(* Logix 5000 project; controller QW361 vendor 1 type 14 code 107 rev 32.11; software revision 32.00; part 13 of 20 *)

        [1807].time.Minute := 9, [1807].time.Second := 59, [1807].time.DST_ON := 1, [1808].log_data[0].min := 1.0, [1808].log_data[0].max := 1.0, [1808].log_data[0].total := 300.0, [1808].log_data[0].time := 300.0, [1808].log_data[0].minminute := 10, [1808].log_data[0].maxminute := 10, [1808].log_data[0].valid := 1, [1808].log_data[1].valid := 1, [1808].log_data[2].valid := 1, [1808].log_data[3].valid := 1, [1808].log_data[4].valid := 1, [1808].time.Year := 2022, [1808].time.Month := 4, [1808].time.Day := 30, [1808].time.Hour := 4, [1808].time.Minute := 14, [1808].time.Second := 59, [1808].time.DST_ON := 1, [1809].log_data[0].min := 1.0, [1809].log_data[0].max := 1.0, [1809].log_data[0].total := 300.0, [1809].log_data[0].time := 300.0, [1809].log_data[0].minminute := 15, [1809].log_data[0].maxminute := 15, [1809].log_data[0].valid := 1, [1809].log_data[1].valid := 1, [1809].log_data[2].valid := 1, [1809].log_data[3].valid := 1, [1809].log_data[4].valid := 1, [1809].time.Year := 2022, [1809].time.Month := 4, [1809].time.Day := 30, [1809].time.Hour := 4, [1809].time.Minute := 19, [1809].time.Second := 59, [1809].time.DST_ON := 1, [1810].log_data[0].min := 1.0, [1810].log_data[0].max := 1.0, [1810].log_data[0].total := 300.0, [1810].log_data[0].time := 300.0, [1810].log_data[0].minminute := 20, [1810].log_data[0].maxminute := 20, [1810].log_data[0].valid := 1, [1810].log_data[1].valid := 1, [1810].log_data[2].valid := 1, [1810].log_data[3].valid := 1, [1810].log_data[4].valid := 1, [1810].time.Year := 2022, [1810].time.Month := 4, [1810].time.Day := 30, [1810].time.Hour := 4, [1810].time.Minute := 24, [1810].time.Second := 59, [1810].time.DST_ON := 1, [1811].log_data[0].min := 1.0, [1811].log_data[0].max := 1.0, [1811].log_data[0].total := 300.0,
        [1811].log_data[0].time := 300.0, [1811].log_data[0].minminute := 25, [1811].log_data[0].maxminute := 25, [1811].log_data[0].valid := 1, [1811].log_data[1].valid := 1, [1811].log_data[2].valid := 1, [1811].log_data[3].valid := 1, [1811].log_data[4].valid := 1, [1811].time.Year := 2022, [1811].time.Month := 4, [1811].time.Day := 30, [1811].time.Hour := 4, [1811].time.Minute := 29, [1811].time.Second := 59, [1811].time.DST_ON := 1, [1812].log_data[0].min := 1.0, [1812].log_data[0].max := 1.0, [1812].log_data[0].total := 300.0, [1812].log_data[0].time := 300.0, [1812].log_data[0].minminute := 30, [1812].log_data[0].maxminute := 30, [1812].log_data[0].valid := 1, [1812].log_data[1].valid := 1, [1812].log_data[2].valid := 1, [1812].log_data[3].valid := 1, [1812].log_data[4].valid := 1, [1812].time.Year := 2022, [1812].time.Month := 4, [1812].time.Day := 30, [1812].time.Hour := 4, [1812].time.Minute := 34, [1812].time.Second := 59, [1812].time.DST_ON := 1, [1813].log_data[0].min := 1.0, [1813].log_data[0].max := 1.0, [1813].log_data[0].total := 300.0, [1813].log_data[0].time := 300.0, [1813].log_data[0].minminute := 35, [1813].log_data[0].maxminute := 35, [1813].log_data[0].valid := 1, [1813].log_data[1].valid := 1, [1813].log_data[2].valid := 1, [1813].log_data[3].valid := 1, [1813].log_data[4].valid := 1, [1813].time.Year := 2022, [1813].time.Month := 4, [1813].time.Day := 30, [1813].time.Hour := 4, [1813].time.Minute := 39, [1813].time.Second := 59, [1813].time.DST_ON := 1, [1814].log_data[0].min := 1.0, [1814].log_data[0].max := 1.0, [1814].log_data[0].total := 300.0, [1814].log_data[0].time := 300.0, [1814].log_data[0].minminute := 40, [1814].log_data[0].maxminute := 40, [1814].log_data[0].valid := 1, [1814].log_data[1].valid := 1, [1814].log_data[2].valid := 1,
        [1814].log_data[3].valid := 1, [1814].log_data[4].valid := 1, [1814].time.Year := 2022, [1814].time.Month := 4, [1814].time.Day := 30, [1814].time.Hour := 4, [1814].time.Minute := 44, [1814].time.Second := 59, [1814].time.DST_ON := 1, [1815].log_data[0].min := 1.0, [1815].log_data[0].max := 1.0, [1815].log_data[0].total := 300.0, [1815].log_data[0].time := 300.0, [1815].log_data[0].minminute := 45, [1815].log_data[0].maxminute := 45, [1815].log_data[0].valid := 1, [1815].log_data[1].valid := 1, [1815].log_data[2].valid := 1, [1815].log_data[3].valid := 1, [1815].log_data[4].valid := 1, [1815].time.Year := 2022, [1815].time.Month := 4, [1815].time.Day := 30, [1815].time.Hour := 4, [1815].time.Minute := 49, [1815].time.Second := 59, [1815].time.DST_ON := 1, [1816].log_data[0].min := 1.0, [1816].log_data[0].max := 1.0, [1816].log_data[0].total := 300.0, [1816].log_data[0].time := 300.0, [1816].log_data[0].minminute := 50, [1816].log_data[0].maxminute := 50, [1816].log_data[0].valid := 1, [1816].log_data[1].valid := 1, [1816].log_data[2].valid := 1, [1816].log_data[3].valid := 1, [1816].log_data[4].valid := 1, [1816].time.Year := 2022, [1816].time.Month := 4, [1816].time.Day := 30, [1816].time.Hour := 4, [1816].time.Minute := 54, [1816].time.Second := 59, [1816].time.DST_ON := 1, [1817].log_data[0].min := 1.0, [1817].log_data[0].max := 1.0, [1817].log_data[0].total := 300.0, [1817].log_data[0].time := 300.0, [1817].log_data[0].minminute := 55, [1817].log_data[0].maxminute := 55, [1817].log_data[0].valid := 1, [1817].log_data[1].valid := 1, [1817].log_data[2].valid := 1, [1817].log_data[3].valid := 1, [1817].log_data[4].valid := 1, [1817].time.Year := 2022, [1817].time.Month := 4, [1817].time.Day := 30, [1817].time.Hour := 4,
        [1817].time.Minute := 59, [1817].time.Second := 59, [1817].time.DST_ON := 1, [1818].log_data[0].min := 1.0, [1818].log_data[0].max := 1.0, [1818].log_data[0].total := 300.0, [1818].log_data[0].time := 300.0, [1818].log_data[0].valid := 1, [1818].log_data[1].valid := 1, [1818].log_data[2].valid := 1, [1818].log_data[3].valid := 1, [1818].log_data[4].valid := 1, [1818].time.Year := 2022, [1818].time.Month := 4, [1818].time.Day := 30, [1818].time.Hour := 5, [1818].time.Minute := 4, [1818].time.Second := 59, [1818].time.DST_ON := 1, [1819].log_data[0].min := 1.0, [1819].log_data[0].max := 1.0, [1819].log_data[0].total := 300.0, [1819].log_data[0].time := 300.0, [1819].log_data[0].minminute := 5, [1819].log_data[0].maxminute := 5, [1819].log_data[0].valid := 1, [1819].log_data[1].valid := 1, [1819].log_data[2].valid := 1, [1819].log_data[3].valid := 1, [1819].log_data[4].valid := 1, [1819].time.Year := 2022, [1819].time.Month := 4, [1819].time.Day := 30, [1819].time.Hour := 5, [1819].time.Minute := 9, [1819].time.Second := 59, [1819].time.DST_ON := 1, [1820].log_data[0].min := 1.0, [1820].log_data[0].max := 1.0, [1820].log_data[0].total := 300.0, [1820].log_data[0].time := 300.0, [1820].log_data[0].minminute := 10, [1820].log_data[0].maxminute := 10, [1820].log_data[0].valid := 1, [1820].log_data[1].valid := 1, [1820].log_data[2].valid := 1, [1820].log_data[3].valid := 1, [1820].log_data[4].valid := 1, [1820].time.Year := 2022, [1820].time.Month := 4, [1820].time.Day := 30, [1820].time.Hour := 5, [1820].time.Minute := 14, [1820].time.Second := 59, [1820].time.DST_ON := 1, [1821].log_data[0].min := 1.0, [1821].log_data[0].max := 1.0, [1821].log_data[0].total := 300.0, [1821].log_data[0].time := 300.0, [1821].log_data[0].minminute := 15,
        [1821].log_data[0].maxminute := 15, [1821].log_data[0].valid := 1, [1821].log_data[1].valid := 1, [1821].log_data[2].valid := 1, [1821].log_data[3].valid := 1, [1821].log_data[4].valid := 1, [1821].time.Year := 2022, [1821].time.Month := 4, [1821].time.Day := 30, [1821].time.Hour := 5, [1821].time.Minute := 19, [1821].time.Second := 59, [1821].time.DST_ON := 1, [1822].log_data[0].min := 1.0, [1822].log_data[0].max := 1.0, [1822].log_data[0].total := 300.0, [1822].log_data[0].time := 300.0, [1822].log_data[0].minminute := 20, [1822].log_data[0].maxminute := 20, [1822].log_data[0].valid := 1, [1822].log_data[1].valid := 1, [1822].log_data[2].valid := 1, [1822].log_data[3].valid := 1, [1822].log_data[4].valid := 1, [1822].time.Year := 2022, [1822].time.Month := 4, [1822].time.Day := 30, [1822].time.Hour := 5, [1822].time.Minute := 24, [1822].time.Second := 59, [1822].time.DST_ON := 1, [1823].log_data[0].min := 1.0, [1823].log_data[0].max := 1.0, [1823].log_data[0].total := 300.0, [1823].log_data[0].time := 300.0, [1823].log_data[0].minminute := 25, [1823].log_data[0].maxminute := 25, [1823].log_data[0].valid := 1, [1823].log_data[1].valid := 1, [1823].log_data[2].valid := 1, [1823].log_data[3].valid := 1, [1823].log_data[4].valid := 1, [1823].time.Year := 2022, [1823].time.Month := 4, [1823].time.Day := 30, [1823].time.Hour := 5, [1823].time.Minute := 29, [1823].time.Second := 59, [1823].time.DST_ON := 1, [1824].log_data[0].min := 1.0, [1824].log_data[0].max := 1.0, [1824].log_data[0].total := 300.0, [1824].log_data[0].time := 300.0, [1824].log_data[0].minminute := 30, [1824].log_data[0].maxminute := 30, [1824].log_data[0].valid := 1, [1824].log_data[1].valid := 1, [1824].log_data[2].valid := 1, [1824].log_data[3].valid := 1, [1824].log_data[4].valid := 1,
        [1824].time.Year := 2022, [1824].time.Month := 4, [1824].time.Day := 30, [1824].time.Hour := 5, [1824].time.Minute := 34, [1824].time.Second := 59, [1824].time.DST_ON := 1, [1825].log_data[0].min := 1.0, [1825].log_data[0].max := 1.0, [1825].log_data[0].total := 300.0, [1825].log_data[0].time := 300.0, [1825].log_data[0].minminute := 35, [1825].log_data[0].maxminute := 35, [1825].log_data[0].valid := 1, [1825].log_data[1].valid := 1, [1825].log_data[2].valid := 1, [1825].log_data[3].valid := 1, [1825].log_data[4].valid := 1, [1825].time.Year := 2022, [1825].time.Month := 4, [1825].time.Day := 30, [1825].time.Hour := 5, [1825].time.Minute := 39, [1825].time.Second := 59, [1825].time.DST_ON := 1, [1826].log_data[0].min := 1.0, [1826].log_data[0].max := 1.0, [1826].log_data[0].total := 300.0, [1826].log_data[0].time := 300.0, [1826].log_data[0].minminute := 40, [1826].log_data[0].maxminute := 40, [1826].log_data[0].valid := 1, [1826].log_data[1].valid := 1, [1826].log_data[2].valid := 1, [1826].log_data[3].valid := 1, [1826].log_data[4].valid := 1, [1826].time.Year := 2022, [1826].time.Month := 4, [1826].time.Day := 30, [1826].time.Hour := 5, [1826].time.Minute := 44, [1826].time.Second := 59, [1826].time.DST_ON := 1, [1827].log_data[0].min := 1.0, [1827].log_data[0].max := 1.0, [1827].log_data[0].total := 299.999, [1827].log_data[0].time := 299.999, [1827].log_data[0].minminute := 45, [1827].log_data[0].maxminute := 45, [1827].log_data[0].valid := 1, [1827].log_data[1].valid := 1, [1827].log_data[2].valid := 1, [1827].log_data[3].valid := 1, [1827].log_data[4].valid := 1, [1827].time.Year := 2022, [1827].time.Month := 4, [1827].time.Day := 30, [1827].time.Hour := 5, [1827].time.Minute := 49, [1827].time.Second := 59,
        [1827].time.DST_ON := 1, [1828].log_data[0].min := 1.0, [1828].log_data[0].max := 1.0, [1828].log_data[0].total := 300.0, [1828].log_data[0].time := 300.0, [1828].log_data[0].minminute := 50, [1828].log_data[0].maxminute := 50, [1828].log_data[0].valid := 1, [1828].log_data[1].valid := 1, [1828].log_data[2].valid := 1, [1828].log_data[3].valid := 1, [1828].log_data[4].valid := 1, [1828].time.Year := 2022, [1828].time.Month := 4, [1828].time.Day := 30, [1828].time.Hour := 5, [1828].time.Minute := 54, [1828].time.Second := 59, [1828].time.DST_ON := 1, [1829].log_data[0].min := 1.0, [1829].log_data[0].max := 1.0, [1829].log_data[0].total := 300.0, [1829].log_data[0].time := 300.0, [1829].log_data[0].minminute := 55, [1829].log_data[0].maxminute := 55, [1829].log_data[0].valid := 1, [1829].log_data[1].valid := 1, [1829].log_data[2].valid := 1, [1829].log_data[3].valid := 1, [1829].log_data[4].valid := 1, [1829].time.Year := 2022, [1829].time.Month := 4, [1829].time.Day := 30, [1829].time.Hour := 5, [1829].time.Minute := 59, [1829].time.Second := 59, [1829].time.DST_ON := 1, [1830].log_data[0].min := 1.0, [1830].log_data[0].max := 1.0, [1830].log_data[0].total := 300.0, [1830].log_data[0].time := 300.0, [1830].log_data[0].valid := 1, [1830].log_data[1].valid := 1, [1830].log_data[2].valid := 1, [1830].log_data[3].valid := 1, [1830].log_data[4].valid := 1, [1830].time.Year := 2022, [1830].time.Month := 4, [1830].time.Day := 30, [1830].time.Hour := 6, [1830].time.Minute := 4, [1830].time.Second := 59, [1830].time.DST_ON := 1, [1831].log_data[0].min := 1.0, [1831].log_data[0].max := 1.0, [1831].log_data[0].total := 300.0, [1831].log_data[0].time := 300.0, [1831].log_data[0].minminute := 5, [1831].log_data[0].maxminute := 5, [1831].log_data[0].valid := 1,
        [1831].log_data[1].valid := 1, [1831].log_data[2].valid := 1, [1831].log_data[3].valid := 1, [1831].log_data[4].valid := 1, [1831].time.Year := 2022, [1831].time.Month := 4, [1831].time.Day := 30, [1831].time.Hour := 6, [1831].time.Minute := 9, [1831].time.Second := 59, [1831].time.DST_ON := 1, [1832].log_data[0].min := 1.0, [1832].log_data[0].max := 1.0, [1832].log_data[0].total := 300.0, [1832].log_data[0].time := 300.0, [1832].log_data[0].minminute := 10, [1832].log_data[0].maxminute := 10, [1832].log_data[0].valid := 1, [1832].log_data[1].valid := 1, [1832].log_data[2].valid := 1, [1832].log_data[3].valid := 1, [1832].log_data[4].valid := 1, [1832].time.Year := 2022, [1832].time.Month := 4, [1832].time.Day := 30, [1832].time.Hour := 6, [1832].time.Minute := 14, [1832].time.Second := 59, [1832].time.DST_ON := 1, [1833].log_data[0].min := 1.0, [1833].log_data[0].max := 1.0, [1833].log_data[0].total := 300.0, [1833].log_data[0].time := 300.0, [1833].log_data[0].minminute := 15, [1833].log_data[0].maxminute := 15, [1833].log_data[0].valid := 1, [1833].log_data[1].valid := 1, [1833].log_data[2].valid := 1, [1833].log_data[3].valid := 1, [1833].log_data[4].valid := 1, [1833].time.Year := 2022, [1833].time.Month := 4, [1833].time.Day := 30, [1833].time.Hour := 6, [1833].time.Minute := 19, [1833].time.Second := 59, [1833].time.DST_ON := 1, [1834].log_data[0].min := 1.0, [1834].log_data[0].max := 1.0, [1834].log_data[0].total := 300.0, [1834].log_data[0].time := 300.0, [1834].log_data[0].minminute := 20, [1834].log_data[0].maxminute := 20, [1834].log_data[0].valid := 1, [1834].log_data[1].valid := 1, [1834].log_data[2].valid := 1, [1834].log_data[3].valid := 1, [1834].log_data[4].valid := 1, [1834].time.Year := 2022, [1834].time.Month := 4,
        [1834].time.Day := 30, [1834].time.Hour := 6, [1834].time.Minute := 24, [1834].time.Second := 59, [1834].time.DST_ON := 1, [1835].log_data[0].min := 1.0, [1835].log_data[0].max := 1.0, [1835].log_data[0].total := 300.0, [1835].log_data[0].time := 300.0, [1835].log_data[0].minminute := 25, [1835].log_data[0].maxminute := 25, [1835].log_data[0].valid := 1, [1835].log_data[1].valid := 1, [1835].log_data[2].valid := 1, [1835].log_data[3].valid := 1, [1835].log_data[4].valid := 1, [1835].time.Year := 2022, [1835].time.Month := 4, [1835].time.Day := 30, [1835].time.Hour := 6, [1835].time.Minute := 29, [1835].time.Second := 59, [1835].time.DST_ON := 1, [1836].log_data[0].min := 1.0, [1836].log_data[0].max := 1.0, [1836].log_data[0].total := 300.0, [1836].log_data[0].time := 300.0, [1836].log_data[0].minminute := 30, [1836].log_data[0].maxminute := 30, [1836].log_data[0].valid := 1, [1836].log_data[1].valid := 1, [1836].log_data[2].valid := 1, [1836].log_data[3].valid := 1, [1836].log_data[4].valid := 1, [1836].time.Year := 2022, [1836].time.Month := 4, [1836].time.Day := 30, [1836].time.Hour := 6, [1836].time.Minute := 34, [1836].time.Second := 59, [1836].time.DST_ON := 1, [1837].log_data[0].min := 1.0, [1837].log_data[0].max := 1.0, [1837].log_data[0].total := 300.0, [1837].log_data[0].time := 300.0, [1837].log_data[0].minminute := 35, [1837].log_data[0].maxminute := 35, [1837].log_data[0].valid := 1, [1837].log_data[1].valid := 1, [1837].log_data[2].valid := 1, [1837].log_data[3].valid := 1, [1837].log_data[4].valid := 1, [1837].time.Year := 2022, [1837].time.Month := 4, [1837].time.Day := 30, [1837].time.Hour := 6, [1837].time.Minute := 39, [1837].time.Second := 59, [1837].time.DST_ON := 1, [1838].log_data[0].min := 1.0,
        [1838].log_data[0].max := 1.0, [1838].log_data[0].total := 300.0, [1838].log_data[0].time := 300.0, [1838].log_data[0].minminute := 40, [1838].log_data[0].maxminute := 40, [1838].log_data[0].valid := 1, [1838].log_data[1].valid := 1, [1838].log_data[2].valid := 1, [1838].log_data[3].valid := 1, [1838].log_data[4].valid := 1, [1838].time.Year := 2022, [1838].time.Month := 4, [1838].time.Day := 30, [1838].time.Hour := 6, [1838].time.Minute := 44, [1838].time.Second := 59, [1838].time.DST_ON := 1, [1839].log_data[0].min := 1.0, [1839].log_data[0].max := 1.0, [1839].log_data[0].total := 300.0, [1839].log_data[0].time := 300.0, [1839].log_data[0].minminute := 45, [1839].log_data[0].maxminute := 45, [1839].log_data[0].valid := 1, [1839].log_data[1].valid := 1, [1839].log_data[2].valid := 1, [1839].log_data[3].valid := 1, [1839].log_data[4].valid := 1, [1839].time.Year := 2022, [1839].time.Month := 4, [1839].time.Day := 30, [1839].time.Hour := 6, [1839].time.Minute := 49, [1839].time.Second := 59, [1839].time.DST_ON := 1, [1840].log_data[0].min := 1.0, [1840].log_data[0].max := 1.0, [1840].log_data[0].total := 300.0, [1840].log_data[0].time := 300.0, [1840].log_data[0].minminute := 50, [1840].log_data[0].maxminute := 50, [1840].log_data[0].valid := 1, [1840].log_data[1].valid := 1, [1840].log_data[2].valid := 1, [1840].log_data[3].valid := 1, [1840].log_data[4].valid := 1, [1840].time.Year := 2022, [1840].time.Month := 4, [1840].time.Day := 30, [1840].time.Hour := 6, [1840].time.Minute := 54, [1840].time.Second := 59, [1840].time.DST_ON := 1, [1841].log_data[0].min := 1.0, [1841].log_data[0].max := 1.0, [1841].log_data[0].total := 300.0, [1841].log_data[0].time := 300.0, [1841].log_data[0].minminute := 55, [1841].log_data[0].maxminute := 55, [1841].log_data[0].valid := 1,
        [1841].log_data[1].valid := 1, [1841].log_data[2].valid := 1, [1841].log_data[3].valid := 1, [1841].log_data[4].valid := 1, [1841].time.Year := 2022, [1841].time.Month := 4, [1841].time.Day := 30, [1841].time.Hour := 6, [1841].time.Minute := 59, [1841].time.Second := 59, [1841].time.DST_ON := 1, [1842].log_data[0].min := 1.0, [1842].log_data[0].max := 1.0, [1842].log_data[0].total := 300.0, [1842].log_data[0].time := 300.0, [1842].log_data[0].valid := 1, [1842].log_data[1].valid := 1, [1842].log_data[2].valid := 1, [1842].log_data[3].valid := 1, [1842].log_data[4].valid := 1, [1842].time.Year := 2022, [1842].time.Month := 4, [1842].time.Day := 30, [1842].time.Hour := 7, [1842].time.Minute := 4, [1842].time.Second := 59, [1842].time.DST_ON := 1, [1843].log_data[0].min := 1.0, [1843].log_data[0].max := 1.0, [1843].log_data[0].total := 300.0, [1843].log_data[0].time := 300.0, [1843].log_data[0].minminute := 5, [1843].log_data[0].maxminute := 5, [1843].log_data[0].valid := 1, [1843].log_data[1].valid := 1, [1843].log_data[2].valid := 1, [1843].log_data[3].valid := 1, [1843].log_data[4].valid := 1, [1843].time.Year := 2022, [1843].time.Month := 4, [1843].time.Day := 30, [1843].time.Hour := 7, [1843].time.Minute := 9, [1843].time.Second := 59, [1843].time.DST_ON := 1, [1844].log_data[0].min := 1.0, [1844].log_data[0].max := 1.0, [1844].log_data[0].total := 300.0, [1844].log_data[0].time := 300.0, [1844].log_data[0].minminute := 10, [1844].log_data[0].maxminute := 10, [1844].log_data[0].valid := 1, [1844].log_data[1].valid := 1, [1844].log_data[2].valid := 1, [1844].log_data[3].valid := 1, [1844].log_data[4].valid := 1, [1844].time.Year := 2022, [1844].time.Month := 4, [1844].time.Day := 30, [1844].time.Hour := 7,
        [1844].time.Minute := 14, [1844].time.Second := 59, [1844].time.DST_ON := 1, [1845].log_data[0].min := 1.0, [1845].log_data[0].max := 1.0, [1845].log_data[0].total := 300.0, [1845].log_data[0].time := 300.0, [1845].log_data[0].minminute := 15, [1845].log_data[0].maxminute := 15, [1845].log_data[0].valid := 1, [1845].log_data[1].valid := 1, [1845].log_data[2].valid := 1, [1845].log_data[3].valid := 1, [1845].log_data[4].valid := 1, [1845].time.Year := 2022, [1845].time.Month := 4, [1845].time.Day := 30, [1845].time.Hour := 7, [1845].time.Minute := 19, [1845].time.Second := 59, [1845].time.DST_ON := 1, [1846].log_data[0].min := 1.0, [1846].log_data[0].max := 1.0, [1846].log_data[0].total := 300.0, [1846].log_data[0].time := 300.0, [1846].log_data[0].minminute := 20, [1846].log_data[0].maxminute := 20, [1846].log_data[0].valid := 1, [1846].log_data[1].valid := 1, [1846].log_data[2].valid := 1, [1846].log_data[3].valid := 1, [1846].log_data[4].valid := 1, [1846].time.Year := 2022, [1846].time.Month := 4, [1846].time.Day := 30, [1846].time.Hour := 7, [1846].time.Minute := 24, [1846].time.Second := 59, [1846].time.DST_ON := 1, [1847].log_data[0].min := 1.0, [1847].log_data[0].max := 1.0, [1847].log_data[0].total := 300.0, [1847].log_data[0].time := 300.0, [1847].log_data[0].minminute := 25, [1847].log_data[0].maxminute := 25, [1847].log_data[0].valid := 1, [1847].log_data[1].valid := 1, [1847].log_data[2].valid := 1, [1847].log_data[3].valid := 1, [1847].log_data[4].valid := 1, [1847].time.Year := 2022, [1847].time.Month := 4, [1847].time.Day := 30, [1847].time.Hour := 7, [1847].time.Minute := 29, [1847].time.Second := 59, [1847].time.DST_ON := 1, [1848].log_data[0].min := 1.0, [1848].log_data[0].max := 1.0, [1848].log_data[0].total := 300.0,
        [1848].log_data[0].time := 300.0, [1848].log_data[0].minminute := 30, [1848].log_data[0].maxminute := 30, [1848].log_data[0].valid := 1, [1848].log_data[1].valid := 1, [1848].log_data[2].valid := 1, [1848].log_data[3].valid := 1, [1848].log_data[4].valid := 1, [1848].time.Year := 2022, [1848].time.Month := 4, [1848].time.Day := 30, [1848].time.Hour := 7, [1848].time.Minute := 34, [1848].time.Second := 59, [1848].time.DST_ON := 1, [1849].log_data[0].min := 1.0, [1849].log_data[0].max := 1.0, [1849].log_data[0].total := 300.0, [1849].log_data[0].time := 300.0, [1849].log_data[0].minminute := 35, [1849].log_data[0].maxminute := 35, [1849].log_data[0].valid := 1, [1849].log_data[1].valid := 1, [1849].log_data[2].valid := 1, [1849].log_data[3].valid := 1, [1849].log_data[4].valid := 1, [1849].time.Year := 2022, [1849].time.Month := 4, [1849].time.Day := 30, [1849].time.Hour := 7, [1849].time.Minute := 39, [1849].time.Second := 59, [1849].time.DST_ON := 1, [1850].log_data[0].min := 1.0, [1850].log_data[0].max := 1.0, [1850].log_data[0].total := 300.0, [1850].log_data[0].time := 300.0, [1850].log_data[0].minminute := 40, [1850].log_data[0].maxminute := 40, [1850].log_data[0].valid := 1, [1850].log_data[1].valid := 1, [1850].log_data[2].valid := 1, [1850].log_data[3].valid := 1, [1850].log_data[4].valid := 1, [1850].time.Year := 2022, [1850].time.Month := 4, [1850].time.Day := 30, [1850].time.Hour := 7, [1850].time.Minute := 44, [1850].time.Second := 59, [1850].time.DST_ON := 1, [1851].log_data[0].min := 1.0, [1851].log_data[0].max := 1.0, [1851].log_data[0].total := 300.0, [1851].log_data[0].time := 300.0, [1851].log_data[0].minminute := 45, [1851].log_data[0].maxminute := 45, [1851].log_data[0].valid := 1, [1851].log_data[1].valid := 1, [1851].log_data[2].valid := 1,
        [1851].log_data[3].valid := 1, [1851].log_data[4].valid := 1, [1851].time.Year := 2022, [1851].time.Month := 4, [1851].time.Day := 30, [1851].time.Hour := 7, [1851].time.Minute := 49, [1851].time.Second := 59, [1851].time.DST_ON := 1, [1852].log_data[0].min := 1.0, [1852].log_data[0].max := 1.0, [1852].log_data[0].total := 300.0, [1852].log_data[0].time := 300.0, [1852].log_data[0].minminute := 50, [1852].log_data[0].maxminute := 50, [1852].log_data[0].valid := 1, [1852].log_data[1].valid := 1, [1852].log_data[2].valid := 1, [1852].log_data[3].valid := 1, [1852].log_data[4].valid := 1, [1852].time.Year := 2022, [1852].time.Month := 4, [1852].time.Day := 30, [1852].time.Hour := 7, [1852].time.Minute := 54, [1852].time.Second := 59, [1852].time.DST_ON := 1, [1853].log_data[0].min := 1.0, [1853].log_data[0].max := 1.0, [1853].log_data[0].total := 300.0, [1853].log_data[0].time := 300.0, [1853].log_data[0].minminute := 55, [1853].log_data[0].maxminute := 55, [1853].log_data[0].valid := 1, [1853].log_data[1].valid := 1, [1853].log_data[2].valid := 1, [1853].log_data[3].valid := 1, [1853].log_data[4].valid := 1, [1853].time.Year := 2022, [1853].time.Month := 4, [1853].time.Day := 30, [1853].time.Hour := 7, [1853].time.Minute := 59, [1853].time.Second := 59, [1853].time.DST_ON := 1, [1854].log_data[0].min := 1.0, [1854].log_data[0].max := 1.0, [1854].log_data[0].total := 300.0, [1854].log_data[0].time := 300.0, [1854].log_data[0].valid := 1, [1854].log_data[1].valid := 1, [1854].log_data[2].valid := 1, [1854].log_data[3].valid := 1, [1854].log_data[4].valid := 1, [1854].time.Year := 2022, [1854].time.Month := 4, [1854].time.Day := 30, [1854].time.Hour := 8, [1854].time.Minute := 4, [1854].time.Second := 59,
        [1854].time.DST_ON := 1, [1855].log_data[0].min := 1.0, [1855].log_data[0].max := 1.0, [1855].log_data[0].total := 300.0, [1855].log_data[0].time := 300.0, [1855].log_data[0].minminute := 5, [1855].log_data[0].maxminute := 5, [1855].log_data[0].valid := 1, [1855].log_data[1].valid := 1, [1855].log_data[2].valid := 1, [1855].log_data[3].valid := 1, [1855].log_data[4].valid := 1, [1855].time.Year := 2022, [1855].time.Month := 4, [1855].time.Day := 30, [1855].time.Hour := 8, [1855].time.Minute := 9, [1855].time.Second := 59, [1855].time.DST_ON := 1, [1856].log_data[0].min := 1.0, [1856].log_data[0].max := 1.0, [1856].log_data[0].total := 300.0, [1856].log_data[0].time := 300.0, [1856].log_data[0].minminute := 10, [1856].log_data[0].maxminute := 10, [1856].log_data[0].valid := 1, [1856].log_data[1].valid := 1, [1856].log_data[2].valid := 1, [1856].log_data[3].valid := 1, [1856].log_data[4].valid := 1, [1856].time.Year := 2022, [1856].time.Month := 4, [1856].time.Day := 30, [1856].time.Hour := 8, [1856].time.Minute := 14, [1856].time.Second := 59, [1856].time.DST_ON := 1, [1857].log_data[0].min := 1.0, [1857].log_data[0].max := 1.0, [1857].log_data[0].total := 299.999, [1857].log_data[0].time := 299.999, [1857].log_data[0].minminute := 15, [1857].log_data[0].maxminute := 15, [1857].log_data[0].valid := 1, [1857].log_data[1].valid := 1, [1857].log_data[2].valid := 1, [1857].log_data[3].valid := 1, [1857].log_data[4].valid := 1, [1857].time.Year := 2022, [1857].time.Month := 4, [1857].time.Day := 30, [1857].time.Hour := 8, [1857].time.Minute := 19, [1857].time.Second := 59, [1857].time.DST_ON := 1, [1858].log_data[0].min := 1.0, [1858].log_data[0].max := 1.0, [1858].log_data[0].total := 300.0, [1858].log_data[0].time := 300.0, [1858].log_data[0].minminute := 20,
        [1858].log_data[0].maxminute := 20, [1858].log_data[0].valid := 1, [1858].log_data[1].valid := 1, [1858].log_data[2].valid := 1, [1858].log_data[3].valid := 1, [1858].log_data[4].valid := 1, [1858].time.Year := 2022, [1858].time.Month := 4, [1858].time.Day := 30, [1858].time.Hour := 8, [1858].time.Minute := 24, [1858].time.Second := 59, [1858].time.DST_ON := 1, [1859].log_data[0].min := 1.0, [1859].log_data[0].max := 1.0, [1859].log_data[0].total := 300.0, [1859].log_data[0].time := 300.0, [1859].log_data[0].minminute := 25, [1859].log_data[0].maxminute := 25, [1859].log_data[0].valid := 1, [1859].log_data[1].valid := 1, [1859].log_data[2].valid := 1, [1859].log_data[3].valid := 1, [1859].log_data[4].valid := 1, [1859].time.Year := 2022, [1859].time.Month := 4, [1859].time.Day := 30, [1859].time.Hour := 8, [1859].time.Minute := 29, [1859].time.Second := 59, [1859].time.DST_ON := 1, [1860].log_data[0].min := 1.0, [1860].log_data[0].max := 1.0, [1860].log_data[0].total := 300.0, [1860].log_data[0].time := 300.0, [1860].log_data[0].minminute := 30, [1860].log_data[0].maxminute := 30, [1860].log_data[0].valid := 1, [1860].log_data[1].valid := 1, [1860].log_data[2].valid := 1, [1860].log_data[3].valid := 1, [1860].log_data[4].valid := 1, [1860].time.Year := 2022, [1860].time.Month := 4, [1860].time.Day := 30, [1860].time.Hour := 8, [1860].time.Minute := 34, [1860].time.Second := 59, [1860].time.DST_ON := 1, [1861].log_data[0].min := 1.0, [1861].log_data[0].max := 1.0, [1861].log_data[0].total := 300.0, [1861].log_data[0].time := 300.0, [1861].log_data[0].minminute := 35, [1861].log_data[0].maxminute := 35, [1861].log_data[0].valid := 1, [1861].log_data[1].valid := 1, [1861].log_data[2].valid := 1, [1861].log_data[3].valid := 1, [1861].log_data[4].valid := 1,
        [1861].time.Year := 2022, [1861].time.Month := 4, [1861].time.Day := 30, [1861].time.Hour := 8, [1861].time.Minute := 39, [1861].time.Second := 59, [1861].time.DST_ON := 1, [1862].log_data[0].min := 1.0, [1862].log_data[0].max := 1.0, [1862].log_data[0].total := 300.0, [1862].log_data[0].time := 300.0, [1862].log_data[0].minminute := 40, [1862].log_data[0].maxminute := 40, [1862].log_data[0].valid := 1, [1862].log_data[1].valid := 1, [1862].log_data[2].valid := 1, [1862].log_data[3].valid := 1, [1862].log_data[4].valid := 1, [1862].time.Year := 2022, [1862].time.Month := 4, [1862].time.Day := 30, [1862].time.Hour := 8, [1862].time.Minute := 44, [1862].time.Second := 59, [1862].time.DST_ON := 1, [1863].log_data[0].min := 1.0, [1863].log_data[0].max := 1.0, [1863].log_data[0].total := 300.0, [1863].log_data[0].time := 300.0, [1863].log_data[0].minminute := 45, [1863].log_data[0].maxminute := 45, [1863].log_data[0].valid := 1, [1863].log_data[1].valid := 1, [1863].log_data[2].valid := 1, [1863].log_data[3].valid := 1, [1863].log_data[4].valid := 1, [1863].time.Year := 2022, [1863].time.Month := 4, [1863].time.Day := 30, [1863].time.Hour := 8, [1863].time.Minute := 49, [1863].time.Second := 59, [1863].time.DST_ON := 1, [1864].log_data[0].min := 1.0, [1864].log_data[0].max := 1.0, [1864].log_data[0].total := 300.0, [1864].log_data[0].time := 300.0, [1864].log_data[0].minminute := 50, [1864].log_data[0].maxminute := 50, [1864].log_data[0].valid := 1, [1864].log_data[1].valid := 1, [1864].log_data[2].valid := 1, [1864].log_data[3].valid := 1, [1864].log_data[4].valid := 1, [1864].time.Year := 2022, [1864].time.Month := 4, [1864].time.Day := 30, [1864].time.Hour := 8, [1864].time.Minute := 54, [1864].time.Second := 59,
        [1864].time.DST_ON := 1, [1865].log_data[0].min := 1.0, [1865].log_data[0].max := 1.0, [1865].log_data[0].total := 300.0, [1865].log_data[0].time := 300.0, [1865].log_data[0].minminute := 55, [1865].log_data[0].maxminute := 55, [1865].log_data[0].valid := 1, [1865].log_data[1].valid := 1, [1865].log_data[2].valid := 1, [1865].log_data[3].valid := 1, [1865].log_data[4].valid := 1, [1865].time.Year := 2022, [1865].time.Month := 4, [1865].time.Day := 30, [1865].time.Hour := 8, [1865].time.Minute := 59, [1865].time.Second := 59, [1865].time.DST_ON := 1, [1866].log_data[0].min := 1.0, [1866].log_data[0].max := 1.0, [1866].log_data[0].total := 300.0, [1866].log_data[0].time := 300.0, [1866].log_data[0].valid := 1, [1866].log_data[1].valid := 1, [1866].log_data[2].valid := 1, [1866].log_data[3].valid := 1, [1866].log_data[4].valid := 1, [1866].time.Year := 2022, [1866].time.Month := 4, [1866].time.Day := 30, [1866].time.Hour := 9, [1866].time.Minute := 4, [1866].time.Second := 59, [1866].time.DST_ON := 1, [1867].log_data[0].min := 1.0, [1867].log_data[0].max := 1.0, [1867].log_data[0].total := 300.0, [1867].log_data[0].time := 300.0, [1867].log_data[0].minminute := 5, [1867].log_data[0].maxminute := 5, [1867].log_data[0].valid := 1, [1867].log_data[1].valid := 1, [1867].log_data[2].valid := 1, [1867].log_data[3].valid := 1, [1867].log_data[4].valid := 1, [1867].time.Year := 2022, [1867].time.Month := 4, [1867].time.Day := 30, [1867].time.Hour := 9, [1867].time.Minute := 9, [1867].time.Second := 59, [1867].time.DST_ON := 1, [1868].log_data[0].min := 1.0, [1868].log_data[0].max := 1.0, [1868].log_data[0].total := 300.0, [1868].log_data[0].time := 300.0, [1868].log_data[0].minminute := 10, [1868].log_data[0].maxminute := 10, [1868].log_data[0].valid := 1,
        [1868].log_data[1].valid := 1, [1868].log_data[2].valid := 1, [1868].log_data[3].valid := 1, [1868].log_data[4].valid := 1, [1868].time.Year := 2022, [1868].time.Month := 4, [1868].time.Day := 30, [1868].time.Hour := 9, [1868].time.Minute := 14, [1868].time.Second := 59, [1868].time.DST_ON := 1, [1869].log_data[0].min := 1.0, [1869].log_data[0].max := 1.0, [1869].log_data[0].total := 300.0, [1869].log_data[0].time := 300.0, [1869].log_data[0].minminute := 15, [1869].log_data[0].maxminute := 15, [1869].log_data[0].valid := 1, [1869].log_data[1].valid := 1, [1869].log_data[2].valid := 1, [1869].log_data[3].valid := 1, [1869].log_data[4].valid := 1, [1869].time.Year := 2022, [1869].time.Month := 4, [1869].time.Day := 30, [1869].time.Hour := 9, [1869].time.Minute := 19, [1869].time.Second := 59, [1869].time.DST_ON := 1, [1870].log_data[0].min := 1.0, [1870].log_data[0].max := 1.0, [1870].log_data[0].total := 300.0, [1870].log_data[0].time := 300.0, [1870].log_data[0].minminute := 20, [1870].log_data[0].maxminute := 20, [1870].log_data[0].valid := 1, [1870].log_data[1].valid := 1, [1870].log_data[2].valid := 1, [1870].log_data[3].valid := 1, [1870].log_data[4].valid := 1, [1870].time.Year := 2022, [1870].time.Month := 4, [1870].time.Day := 30, [1870].time.Hour := 9, [1870].time.Minute := 24, [1870].time.Second := 59, [1870].time.DST_ON := 1, [1871].log_data[0].min := 1.0, [1871].log_data[0].max := 1.0, [1871].log_data[0].total := 300.0, [1871].log_data[0].time := 300.0, [1871].log_data[0].minminute := 25, [1871].log_data[0].maxminute := 25, [1871].log_data[0].valid := 1, [1871].log_data[1].valid := 1, [1871].log_data[2].valid := 1, [1871].log_data[3].valid := 1, [1871].log_data[4].valid := 1, [1871].time.Year := 2022, [1871].time.Month := 4,
        [1871].time.Day := 30, [1871].time.Hour := 9, [1871].time.Minute := 29, [1871].time.Second := 59, [1871].time.DST_ON := 1, [1872].log_data[0].min := 1.0, [1872].log_data[0].max := 1.0, [1872].log_data[0].total := 300.0, [1872].log_data[0].time := 300.0, [1872].log_data[0].minminute := 30, [1872].log_data[0].maxminute := 30, [1872].log_data[0].valid := 1, [1872].log_data[1].valid := 1, [1872].log_data[2].valid := 1, [1872].log_data[3].valid := 1, [1872].log_data[4].valid := 1, [1872].time.Year := 2022, [1872].time.Month := 4, [1872].time.Day := 30, [1872].time.Hour := 9, [1872].time.Minute := 34, [1872].time.Second := 59, [1872].time.DST_ON := 1, [1873].log_data[0].min := 1.0, [1873].log_data[0].max := 1.0, [1873].log_data[0].total := 300.0, [1873].log_data[0].time := 300.0, [1873].log_data[0].minminute := 35, [1873].log_data[0].maxminute := 35, [1873].log_data[0].valid := 1, [1873].log_data[1].valid := 1, [1873].log_data[2].valid := 1, [1873].log_data[3].valid := 1, [1873].log_data[4].valid := 1, [1873].time.Year := 2022, [1873].time.Month := 4, [1873].time.Day := 30, [1873].time.Hour := 9, [1873].time.Minute := 39, [1873].time.Second := 59, [1873].time.DST_ON := 1, [1874].log_data[0].min := 1.0, [1874].log_data[0].max := 1.0, [1874].log_data[0].total := 300.0, [1874].log_data[0].time := 300.0, [1874].log_data[0].minminute := 40, [1874].log_data[0].maxminute := 40, [1874].log_data[0].valid := 1, [1874].log_data[1].valid := 1, [1874].log_data[2].valid := 1, [1874].log_data[3].valid := 1, [1874].log_data[4].valid := 1, [1874].time.Year := 2022, [1874].time.Month := 4, [1874].time.Day := 30, [1874].time.Hour := 9, [1874].time.Minute := 44, [1874].time.Second := 59, [1874].time.DST_ON := 1, [1875].log_data[0].min := 1.0,
        [1875].log_data[0].max := 1.0, [1875].log_data[0].total := 300.0, [1875].log_data[0].time := 300.0, [1875].log_data[0].minminute := 45, [1875].log_data[0].maxminute := 45, [1875].log_data[0].valid := 1, [1875].log_data[1].valid := 1, [1875].log_data[2].valid := 1, [1875].log_data[3].valid := 1, [1875].log_data[4].valid := 1, [1875].time.Year := 2022, [1875].time.Month := 4, [1875].time.Day := 30, [1875].time.Hour := 9, [1875].time.Minute := 49, [1875].time.Second := 59, [1875].time.DST_ON := 1, [1876].log_data[0].min := 1.0, [1876].log_data[0].max := 1.0, [1876].log_data[0].total := 300.0, [1876].log_data[0].time := 300.0, [1876].log_data[0].minminute := 50, [1876].log_data[0].maxminute := 50, [1876].log_data[0].valid := 1, [1876].log_data[1].valid := 1, [1876].log_data[2].valid := 1, [1876].log_data[3].valid := 1, [1876].log_data[4].valid := 1, [1876].time.Year := 2022, [1876].time.Month := 4, [1876].time.Day := 30, [1876].time.Hour := 9, [1876].time.Minute := 54, [1876].time.Second := 59, [1876].time.DST_ON := 1, [1877].log_data[0].min := 1.0, [1877].log_data[0].max := 1.0, [1877].log_data[0].total := 300.0, [1877].log_data[0].time := 300.0, [1877].log_data[0].minminute := 55, [1877].log_data[0].maxminute := 55, [1877].log_data[0].valid := 1, [1877].log_data[1].valid := 1, [1877].log_data[2].valid := 1, [1877].log_data[3].valid := 1, [1877].log_data[4].valid := 1, [1877].time.Year := 2022, [1877].time.Month := 4, [1877].time.Day := 30, [1877].time.Hour := 9, [1877].time.Minute := 59, [1877].time.Second := 59, [1877].time.DST_ON := 1, [1878].log_data[0].min := 1.0, [1878].log_data[0].max := 1.0, [1878].log_data[0].total := 300.0, [1878].log_data[0].time := 300.0, [1878].log_data[0].valid := 1, [1878].log_data[1].valid := 1, [1878].log_data[2].valid := 1,
        [1878].log_data[3].valid := 1, [1878].log_data[4].valid := 1, [1878].time.Year := 2022, [1878].time.Month := 4, [1878].time.Day := 30, [1878].time.Hour := 10, [1878].time.Minute := 4, [1878].time.Second := 59, [1878].time.DST_ON := 1, [1879].log_data[0].min := 1.0, [1879].log_data[0].max := 1.0, [1879].log_data[0].total := 300.0, [1879].log_data[0].time := 300.0, [1879].log_data[0].minminute := 5, [1879].log_data[0].maxminute := 5, [1879].log_data[0].valid := 1, [1879].log_data[1].valid := 1, [1879].log_data[2].valid := 1, [1879].log_data[3].valid := 1, [1879].log_data[4].valid := 1, [1879].time.Year := 2022, [1879].time.Month := 4, [1879].time.Day := 30, [1879].time.Hour := 10, [1879].time.Minute := 9, [1879].time.Second := 59, [1879].time.DST_ON := 1, [1880].log_data[0].min := 1.0, [1880].log_data[0].max := 1.0, [1880].log_data[0].total := 300.0, [1880].log_data[0].time := 300.0, [1880].log_data[0].minminute := 10, [1880].log_data[0].maxminute := 10, [1880].log_data[0].valid := 1, [1880].log_data[1].valid := 1, [1880].log_data[2].valid := 1, [1880].log_data[3].valid := 1, [1880].log_data[4].valid := 1, [1880].time.Year := 2022, [1880].time.Month := 4, [1880].time.Day := 30, [1880].time.Hour := 10, [1880].time.Minute := 14, [1880].time.Second := 59, [1880].time.DST_ON := 1, [1881].log_data[0].min := 1.0, [1881].log_data[0].max := 1.0, [1881].log_data[0].total := 300.0, [1881].log_data[0].time := 300.0, [1881].log_data[0].minminute := 15, [1881].log_data[0].maxminute := 15, [1881].log_data[0].valid := 1, [1881].log_data[1].valid := 1, [1881].log_data[2].valid := 1, [1881].log_data[3].valid := 1, [1881].log_data[4].valid := 1, [1881].time.Year := 2022, [1881].time.Month := 4, [1881].time.Day := 30, [1881].time.Hour := 10,
        [1881].time.Minute := 19, [1881].time.Second := 59, [1881].time.DST_ON := 1, [1882].log_data[0].min := 1.0, [1882].log_data[0].max := 1.0, [1882].log_data[0].total := 300.0, [1882].log_data[0].time := 300.0, [1882].log_data[0].minminute := 20, [1882].log_data[0].maxminute := 20, [1882].log_data[0].valid := 1, [1882].log_data[1].valid := 1, [1882].log_data[2].valid := 1, [1882].log_data[3].valid := 1, [1882].log_data[4].valid := 1, [1882].time.Year := 2022, [1882].time.Month := 4, [1882].time.Day := 30, [1882].time.Hour := 10, [1882].time.Minute := 24, [1882].time.Second := 59, [1882].time.DST_ON := 1, [1883].log_data[0].min := 1.0, [1883].log_data[0].max := 1.0, [1883].log_data[0].total := 300.0, [1883].log_data[0].time := 300.0, [1883].log_data[0].minminute := 25, [1883].log_data[0].maxminute := 25, [1883].log_data[0].valid := 1, [1883].log_data[1].valid := 1, [1883].log_data[2].valid := 1, [1883].log_data[3].valid := 1, [1883].log_data[4].valid := 1, [1883].time.Year := 2022, [1883].time.Month := 4, [1883].time.Day := 30, [1883].time.Hour := 10, [1883].time.Minute := 29, [1883].time.Second := 59, [1883].time.DST_ON := 1, [1884].log_data[0].min := 1.0, [1884].log_data[0].max := 1.0, [1884].log_data[0].total := 300.0, [1884].log_data[0].time := 300.0, [1884].log_data[0].minminute := 30, [1884].log_data[0].maxminute := 30, [1884].log_data[0].valid := 1, [1884].log_data[1].valid := 1, [1884].log_data[2].valid := 1, [1884].log_data[3].valid := 1, [1884].log_data[4].valid := 1, [1884].time.Year := 2022, [1884].time.Month := 4, [1884].time.Day := 30, [1884].time.Hour := 10, [1884].time.Minute := 34, [1884].time.Second := 59, [1884].time.DST_ON := 1, [1885].log_data[0].min := 1.0, [1885].log_data[0].max := 1.0, [1885].log_data[0].total := 300.0,
        [1885].log_data[0].time := 300.0, [1885].log_data[0].minminute := 35, [1885].log_data[0].maxminute := 35, [1885].log_data[0].valid := 1, [1885].log_data[1].valid := 1, [1885].log_data[2].valid := 1, [1885].log_data[3].valid := 1, [1885].log_data[4].valid := 1, [1885].time.Year := 2022, [1885].time.Month := 4, [1885].time.Day := 30, [1885].time.Hour := 10, [1885].time.Minute := 39, [1885].time.Second := 59, [1885].time.DST_ON := 1, [1886].log_data[0].min := 1.0, [1886].log_data[0].max := 1.0, [1886].log_data[0].total := 300.0, [1886].log_data[0].time := 300.0, [1886].log_data[0].minminute := 40, [1886].log_data[0].maxminute := 40, [1886].log_data[0].valid := 1, [1886].log_data[1].valid := 1, [1886].log_data[2].valid := 1, [1886].log_data[3].valid := 1, [1886].log_data[4].valid := 1, [1886].time.Year := 2022, [1886].time.Month := 4, [1886].time.Day := 30, [1886].time.Hour := 10, [1886].time.Minute := 44, [1886].time.Second := 59, [1886].time.DST_ON := 1, [1887].log_data[0].min := 1.0, [1887].log_data[0].max := 1.0, [1887].log_data[0].total := 300.0, [1887].log_data[0].time := 300.0, [1887].log_data[0].minminute := 45, [1887].log_data[0].maxminute := 45, [1887].log_data[0].valid := 1, [1887].log_data[1].valid := 1, [1887].log_data[2].valid := 1, [1887].log_data[3].valid := 1, [1887].log_data[4].valid := 1, [1887].time.Year := 2022, [1887].time.Month := 4, [1887].time.Day := 30, [1887].time.Hour := 10, [1887].time.Minute := 49, [1887].time.Second := 59, [1887].time.DST_ON := 1, [1888].log_data[0].min := 1.0, [1888].log_data[0].max := 1.0, [1888].log_data[0].total := 300.0, [1888].log_data[0].time := 300.0, [1888].log_data[0].minminute := 50, [1888].log_data[0].maxminute := 50, [1888].log_data[0].valid := 1, [1888].log_data[1].valid := 1, [1888].log_data[2].valid := 1,
        [1888].log_data[3].valid := 1, [1888].log_data[4].valid := 1, [1888].time.Year := 2022, [1888].time.Month := 4, [1888].time.Day := 30, [1888].time.Hour := 10, [1888].time.Minute := 54, [1888].time.Second := 59, [1888].time.DST_ON := 1, [1889].log_data[0].min := 1.0, [1889].log_data[0].max := 1.0, [1889].log_data[0].total := 300.0, [1889].log_data[0].time := 300.0, [1889].log_data[0].minminute := 55, [1889].log_data[0].maxminute := 55, [1889].log_data[0].valid := 1, [1889].log_data[1].valid := 1, [1889].log_data[2].valid := 1, [1889].log_data[3].valid := 1, [1889].log_data[4].valid := 1, [1889].time.Year := 2022, [1889].time.Month := 4, [1889].time.Day := 30, [1889].time.Hour := 10, [1889].time.Minute := 59, [1889].time.Second := 59, [1889].time.DST_ON := 1, [1890].log_data[0].min := 1.0, [1890].log_data[0].max := 1.0, [1890].log_data[0].total := 300.0, [1890].log_data[0].time := 300.0, [1890].log_data[0].valid := 1, [1890].log_data[1].valid := 1, [1890].log_data[2].valid := 1, [1890].log_data[3].valid := 1, [1890].log_data[4].valid := 1, [1890].time.Year := 2022, [1890].time.Month := 4, [1890].time.Day := 30, [1890].time.Hour := 11, [1890].time.Minute := 4, [1890].time.Second := 59, [1890].time.DST_ON := 1, [1891].log_data[0].min := 1.0, [1891].log_data[0].max := 1.0, [1891].log_data[0].total := 300.0, [1891].log_data[0].time := 300.0, [1891].log_data[0].minminute := 5, [1891].log_data[0].maxminute := 5, [1891].log_data[0].valid := 1, [1891].log_data[1].valid := 1, [1891].log_data[2].valid := 1, [1891].log_data[3].valid := 1, [1891].log_data[4].valid := 1, [1891].time.Year := 2022, [1891].time.Month := 4, [1891].time.Day := 30, [1891].time.Hour := 11, [1891].time.Minute := 9, [1891].time.Second := 59,
        [1891].time.DST_ON := 1, [1892].log_data[0].min := 1.0, [1892].log_data[0].max := 1.0, [1892].log_data[0].total := 300.0, [1892].log_data[0].time := 300.0, [1892].log_data[0].minminute := 10, [1892].log_data[0].maxminute := 10, [1892].log_data[0].valid := 1, [1892].log_data[1].valid := 1, [1892].log_data[2].valid := 1, [1892].log_data[3].valid := 1, [1892].log_data[4].valid := 1, [1892].time.Year := 2022, [1892].time.Month := 4, [1892].time.Day := 30, [1892].time.Hour := 11, [1892].time.Minute := 14, [1892].time.Second := 59, [1892].time.DST_ON := 1, [1893].log_data[0].min := 1.0, [1893].log_data[0].max := 1.0, [1893].log_data[0].total := 300.0, [1893].log_data[0].time := 300.0, [1893].log_data[0].minminute := 15, [1893].log_data[0].maxminute := 15, [1893].log_data[0].valid := 1, [1893].log_data[1].valid := 1, [1893].log_data[2].valid := 1, [1893].log_data[3].valid := 1, [1893].log_data[4].valid := 1, [1893].time.Year := 2022, [1893].time.Month := 4, [1893].time.Day := 30, [1893].time.Hour := 11, [1893].time.Minute := 19, [1893].time.Second := 59, [1893].time.DST_ON := 1, [1894].log_data[0].min := 1.0, [1894].log_data[0].max := 1.0, [1894].log_data[0].total := 300.0, [1894].log_data[0].time := 300.0, [1894].log_data[0].minminute := 20, [1894].log_data[0].maxminute := 20, [1894].log_data[0].valid := 1, [1894].log_data[1].valid := 1, [1894].log_data[2].valid := 1, [1894].log_data[3].valid := 1, [1894].log_data[4].valid := 1, [1894].time.Year := 2022, [1894].time.Month := 4, [1894].time.Day := 30, [1894].time.Hour := 11, [1894].time.Minute := 24, [1894].time.Second := 59, [1894].time.DST_ON := 1, [1895].log_data[0].min := 1.0, [1895].log_data[0].max := 1.0, [1895].log_data[0].total := 300.0, [1895].log_data[0].time := 300.0, [1895].log_data[0].minminute := 25,
        [1895].log_data[0].maxminute := 25, [1895].log_data[0].valid := 1, [1895].log_data[1].valid := 1, [1895].log_data[2].valid := 1, [1895].log_data[3].valid := 1, [1895].log_data[4].valid := 1, [1895].time.Year := 2022, [1895].time.Month := 4, [1895].time.Day := 30, [1895].time.Hour := 11, [1895].time.Minute := 29, [1895].time.Second := 59, [1895].time.DST_ON := 1, [1896].log_data[0].min := 1.0, [1896].log_data[0].max := 1.0, [1896].log_data[0].total := 300.0, [1896].log_data[0].time := 300.0, [1896].log_data[0].minminute := 30, [1896].log_data[0].maxminute := 30, [1896].log_data[0].valid := 1, [1896].log_data[1].valid := 1, [1896].log_data[2].valid := 1, [1896].log_data[3].valid := 1, [1896].log_data[4].valid := 1, [1896].time.Year := 2022, [1896].time.Month := 4, [1896].time.Day := 30, [1896].time.Hour := 11, [1896].time.Minute := 34, [1896].time.Second := 59, [1896].time.DST_ON := 1, [1897].log_data[0].min := 1.0, [1897].log_data[0].max := 1.0, [1897].log_data[0].total := 300.0, [1897].log_data[0].time := 300.0, [1897].log_data[0].minminute := 35, [1897].log_data[0].maxminute := 35, [1897].log_data[0].valid := 1, [1897].log_data[1].valid := 1, [1897].log_data[2].valid := 1, [1897].log_data[3].valid := 1, [1897].log_data[4].valid := 1, [1897].time.Year := 2022, [1897].time.Month := 4, [1897].time.Day := 30, [1897].time.Hour := 11, [1897].time.Minute := 39, [1897].time.Second := 59, [1897].time.DST_ON := 1, [1898].log_data[0].min := 1.0, [1898].log_data[0].max := 1.0, [1898].log_data[0].total := 300.0, [1898].log_data[0].time := 300.0, [1898].log_data[0].minminute := 40, [1898].log_data[0].maxminute := 40, [1898].log_data[0].valid := 1, [1898].log_data[1].valid := 1, [1898].log_data[2].valid := 1, [1898].log_data[3].valid := 1, [1898].log_data[4].valid := 1,
        [1898].time.Year := 2022, [1898].time.Month := 4, [1898].time.Day := 30, [1898].time.Hour := 11, [1898].time.Minute := 44, [1898].time.Second := 59, [1898].time.DST_ON := 1, [1899].log_data[0].min := 1.0, [1899].log_data[0].max := 1.0, [1899].log_data[0].total := 300.0, [1899].log_data[0].time := 300.0, [1899].log_data[0].minminute := 45, [1899].log_data[0].maxminute := 45, [1899].log_data[0].valid := 1, [1899].log_data[1].valid := 1, [1899].log_data[2].valid := 1, [1899].log_data[3].valid := 1, [1899].log_data[4].valid := 1, [1899].time.Year := 2022, [1899].time.Month := 4, [1899].time.Day := 30, [1899].time.Hour := 11, [1899].time.Minute := 49, [1899].time.Second := 59, [1899].time.DST_ON := 1, [1900].log_data[0].min := 1.0, [1900].log_data[0].max := 1.0, [1900].log_data[0].total := 300.001, [1900].log_data[0].time := 300.001, [1900].log_data[0].minminute := 50, [1900].log_data[0].maxminute := 50, [1900].log_data[0].valid := 1, [1900].log_data[1].valid := 1, [1900].log_data[2].valid := 1, [1900].log_data[3].valid := 1, [1900].log_data[4].valid := 1, [1900].time.Year := 2022, [1900].time.Month := 4, [1900].time.Day := 30, [1900].time.Hour := 11, [1900].time.Minute := 54, [1900].time.Second := 59, [1900].time.DST_ON := 1, [1901].log_data[0].min := 1.0, [1901].log_data[0].max := 1.0, [1901].log_data[0].total := 300.0, [1901].log_data[0].time := 300.0, [1901].log_data[0].minminute := 55, [1901].log_data[0].maxminute := 55, [1901].log_data[0].valid := 1, [1901].log_data[1].valid := 1, [1901].log_data[2].valid := 1, [1901].log_data[3].valid := 1, [1901].log_data[4].valid := 1, [1901].time.Year := 2022, [1901].time.Month := 4, [1901].time.Day := 30, [1901].time.Hour := 11, [1901].time.Minute := 59, [1901].time.Second := 59,
        [1901].time.DST_ON := 1, [1902].log_data[0].min := 1.0, [1902].log_data[0].max := 1.0, [1902].log_data[0].total := 300.0, [1902].log_data[0].time := 300.0, [1902].log_data[0].valid := 1, [1902].log_data[1].valid := 1, [1902].log_data[2].valid := 1, [1902].log_data[3].valid := 1, [1902].log_data[4].valid := 1, [1902].time.Year := 2022, [1902].time.Month := 4, [1902].time.Day := 30, [1902].time.Hour := 12, [1902].time.Minute := 4, [1902].time.Second := 59, [1902].time.DST_ON := 1, [1903].log_data[0].min := 1.0, [1903].log_data[0].max := 1.0, [1903].log_data[0].total := 300.0, [1903].log_data[0].time := 300.0, [1903].log_data[0].minminute := 5, [1903].log_data[0].maxminute := 5, [1903].log_data[0].valid := 1, [1903].log_data[1].valid := 1, [1903].log_data[2].valid := 1, [1903].log_data[3].valid := 1, [1903].log_data[4].valid := 1, [1903].time.Year := 2022, [1903].time.Month := 4, [1903].time.Day := 30, [1903].time.Hour := 12, [1903].time.Minute := 9, [1903].time.Second := 59, [1903].time.DST_ON := 1, [1904].log_data[0].min := 1.0, [1904].log_data[0].max := 1.0, [1904].log_data[0].total := 300.0, [1904].log_data[0].time := 300.0, [1904].log_data[0].minminute := 10, [1904].log_data[0].maxminute := 10, [1904].log_data[0].valid := 1, [1904].log_data[1].valid := 1, [1904].log_data[2].valid := 1, [1904].log_data[3].valid := 1, [1904].log_data[4].valid := 1, [1904].time.Year := 2022, [1904].time.Month := 4, [1904].time.Day := 30, [1904].time.Hour := 12, [1904].time.Minute := 14, [1904].time.Second := 59, [1904].time.DST_ON := 1, [1905].log_data[0].min := 1.0, [1905].log_data[0].max := 1.0, [1905].log_data[0].total := 300.0, [1905].log_data[0].time := 300.0, [1905].log_data[0].minminute := 15, [1905].log_data[0].maxminute := 15, [1905].log_data[0].valid := 1,
        [1905].log_data[1].valid := 1, [1905].log_data[2].valid := 1, [1905].log_data[3].valid := 1, [1905].log_data[4].valid := 1, [1905].time.Year := 2022, [1905].time.Month := 4, [1905].time.Day := 30, [1905].time.Hour := 12, [1905].time.Minute := 19, [1905].time.Second := 59, [1905].time.DST_ON := 1, [1906].log_data[0].min := 1.0, [1906].log_data[0].max := 1.0, [1906].log_data[0].total := 300.0, [1906].log_data[0].time := 300.0, [1906].log_data[0].minminute := 20, [1906].log_data[0].maxminute := 20, [1906].log_data[0].valid := 1, [1906].log_data[1].valid := 1, [1906].log_data[2].valid := 1, [1906].log_data[3].valid := 1, [1906].log_data[4].valid := 1, [1906].time.Year := 2022, [1906].time.Month := 4, [1906].time.Day := 30, [1906].time.Hour := 12, [1906].time.Minute := 24, [1906].time.Second := 59, [1906].time.DST_ON := 1, [1907].log_data[0].min := 1.0, [1907].log_data[0].max := 1.0, [1907].log_data[0].total := 300.0, [1907].log_data[0].time := 300.0, [1907].log_data[0].minminute := 25, [1907].log_data[0].maxminute := 25, [1907].log_data[0].valid := 1, [1907].log_data[1].valid := 1, [1907].log_data[2].valid := 1, [1907].log_data[3].valid := 1, [1907].log_data[4].valid := 1, [1907].time.Year := 2022, [1907].time.Month := 4, [1907].time.Day := 30, [1907].time.Hour := 12, [1907].time.Minute := 29, [1907].time.Second := 59, [1907].time.DST_ON := 1, [1908].log_data[0].min := 1.0, [1908].log_data[0].max := 1.0, [1908].log_data[0].total := 300.0, [1908].log_data[0].time := 300.0, [1908].log_data[0].minminute := 30, [1908].log_data[0].maxminute := 30, [1908].log_data[0].valid := 1, [1908].log_data[1].valid := 1, [1908].log_data[2].valid := 1, [1908].log_data[3].valid := 1, [1908].log_data[4].valid := 1, [1908].time.Year := 2022, [1908].time.Month := 4,
        [1908].time.Day := 30, [1908].time.Hour := 12, [1908].time.Minute := 34, [1908].time.Second := 59, [1908].time.DST_ON := 1, [1909].log_data[0].min := 1.0, [1909].log_data[0].max := 1.0, [1909].log_data[0].total := 300.0, [1909].log_data[0].time := 300.0, [1909].log_data[0].minminute := 35, [1909].log_data[0].maxminute := 35, [1909].log_data[0].valid := 1, [1909].log_data[1].valid := 1, [1909].log_data[2].valid := 1, [1909].log_data[3].valid := 1, [1909].log_data[4].valid := 1, [1909].time.Year := 2022, [1909].time.Month := 4, [1909].time.Day := 30, [1909].time.Hour := 12, [1909].time.Minute := 39, [1909].time.Second := 59, [1909].time.DST_ON := 1, [1910].log_data[0].min := 1.0, [1910].log_data[0].max := 1.0, [1910].log_data[0].total := 299.999, [1910].log_data[0].time := 299.999, [1910].log_data[0].minminute := 40, [1910].log_data[0].maxminute := 40, [1910].log_data[0].valid := 1, [1910].log_data[1].valid := 1, [1910].log_data[2].valid := 1, [1910].log_data[3].valid := 1, [1910].log_data[4].valid := 1, [1910].time.Year := 2022, [1910].time.Month := 4, [1910].time.Day := 30, [1910].time.Hour := 12, [1910].time.Minute := 44, [1910].time.Second := 59, [1910].time.DST_ON := 1, [1911].log_data[0].min := 1.0, [1911].log_data[0].max := 1.0, [1911].log_data[0].total := 300.0, [1911].log_data[0].time := 300.0, [1911].log_data[0].minminute := 45, [1911].log_data[0].maxminute := 45, [1911].log_data[0].valid := 1, [1911].log_data[1].valid := 1, [1911].log_data[2].valid := 1, [1911].log_data[3].valid := 1, [1911].log_data[4].valid := 1, [1911].time.Year := 2022, [1911].time.Month := 4, [1911].time.Day := 30, [1911].time.Hour := 12, [1911].time.Minute := 49, [1911].time.Second := 59, [1911].time.DST_ON := 1, [1912].log_data[0].min := 1.0,
        [1912].log_data[0].max := 1.0, [1912].log_data[0].total := 300.0, [1912].log_data[0].time := 300.0, [1912].log_data[0].minminute := 50, [1912].log_data[0].maxminute := 50, [1912].log_data[0].valid := 1, [1912].log_data[1].valid := 1, [1912].log_data[2].valid := 1, [1912].log_data[3].valid := 1, [1912].log_data[4].valid := 1, [1912].time.Year := 2022, [1912].time.Month := 4, [1912].time.Day := 30, [1912].time.Hour := 12, [1912].time.Minute := 54, [1912].time.Second := 59, [1912].time.DST_ON := 1, [1913].log_data[0].min := 1.0, [1913].log_data[0].max := 1.0, [1913].log_data[0].total := 300.0, [1913].log_data[0].time := 300.0, [1913].log_data[0].minminute := 55, [1913].log_data[0].maxminute := 55, [1913].log_data[0].valid := 1, [1913].log_data[1].valid := 1, [1913].log_data[2].valid := 1, [1913].log_data[3].valid := 1, [1913].log_data[4].valid := 1, [1913].time.Year := 2022, [1913].time.Month := 4, [1913].time.Day := 30, [1913].time.Hour := 12, [1913].time.Minute := 59, [1913].time.Second := 59, [1913].time.DST_ON := 1, [1914].log_data[0].min := 1.0, [1914].log_data[0].max := 1.0, [1914].log_data[0].total := 300.0, [1914].log_data[0].time := 300.0, [1914].log_data[0].valid := 1, [1914].log_data[1].valid := 1, [1914].log_data[2].valid := 1, [1914].log_data[3].valid := 1, [1914].log_data[4].valid := 1, [1914].time.Year := 2022, [1914].time.Month := 4, [1914].time.Day := 30, [1914].time.Hour := 13, [1914].time.Minute := 4, [1914].time.Second := 59, [1914].time.DST_ON := 1, [1915].log_data[0].min := 1.0, [1915].log_data[0].max := 1.0, [1915].log_data[0].total := 300.0, [1915].log_data[0].time := 300.0, [1915].log_data[0].minminute := 5, [1915].log_data[0].maxminute := 5, [1915].log_data[0].valid := 1, [1915].log_data[1].valid := 1, [1915].log_data[2].valid := 1,
        [1915].log_data[3].valid := 1, [1915].log_data[4].valid := 1, [1915].time.Year := 2022, [1915].time.Month := 4, [1915].time.Day := 30, [1915].time.Hour := 13, [1915].time.Minute := 9, [1915].time.Second := 59, [1915].time.DST_ON := 1, [1916].log_data[0].min := 1.0, [1916].log_data[0].max := 1.0, [1916].log_data[0].total := 300.0, [1916].log_data[0].time := 300.0, [1916].log_data[0].minminute := 10, [1916].log_data[0].maxminute := 10, [1916].log_data[0].valid := 1, [1916].log_data[1].valid := 1, [1916].log_data[2].valid := 1, [1916].log_data[3].valid := 1, [1916].log_data[4].valid := 1, [1916].time.Year := 2022, [1916].time.Month := 4, [1916].time.Day := 30, [1916].time.Hour := 13, [1916].time.Minute := 14, [1916].time.Second := 59, [1916].time.DST_ON := 1, [1917].log_data[0].min := 1.0, [1917].log_data[0].max := 1.0, [1917].log_data[0].total := 300.0, [1917].log_data[0].time := 300.0, [1917].log_data[0].minminute := 15, [1917].log_data[0].maxminute := 15, [1917].log_data[0].valid := 1, [1917].log_data[1].valid := 1, [1917].log_data[2].valid := 1, [1917].log_data[3].valid := 1, [1917].log_data[4].valid := 1, [1917].time.Year := 2022, [1917].time.Month := 4, [1917].time.Day := 30, [1917].time.Hour := 13, [1917].time.Minute := 19, [1917].time.Second := 59, [1917].time.DST_ON := 1, [1918].log_data[0].min := 1.0, [1918].log_data[0].max := 1.0, [1918].log_data[0].total := 300.0, [1918].log_data[0].time := 300.0, [1918].log_data[0].minminute := 20, [1918].log_data[0].maxminute := 20, [1918].log_data[0].valid := 1, [1918].log_data[1].valid := 1, [1918].log_data[2].valid := 1, [1918].log_data[3].valid := 1, [1918].log_data[4].valid := 1, [1918].time.Year := 2022, [1918].time.Month := 4, [1918].time.Day := 30, [1918].time.Hour := 13,
        [1918].time.Minute := 24, [1918].time.Second := 59, [1918].time.DST_ON := 1, [1919].log_data[0].min := 1.0, [1919].log_data[0].max := 1.0, [1919].log_data[0].total := 300.0, [1919].log_data[0].time := 300.0, [1919].log_data[0].minminute := 25, [1919].log_data[0].maxminute := 25, [1919].log_data[0].valid := 1, [1919].log_data[1].valid := 1, [1919].log_data[2].valid := 1, [1919].log_data[3].valid := 1, [1919].log_data[4].valid := 1, [1919].time.Year := 2022, [1919].time.Month := 4, [1919].time.Day := 30, [1919].time.Hour := 13, [1919].time.Minute := 29, [1919].time.Second := 59, [1919].time.DST_ON := 1, [1920].log_data[0].min := 1.0, [1920].log_data[0].max := 1.0, [1920].log_data[0].total := 300.0, [1920].log_data[0].time := 300.0, [1920].log_data[0].minminute := 30, [1920].log_data[0].maxminute := 30, [1920].log_data[0].valid := 1, [1920].log_data[1].valid := 1, [1920].log_data[2].valid := 1, [1920].log_data[3].valid := 1, [1920].log_data[4].valid := 1, [1920].time.Year := 2022, [1920].time.Month := 4, [1920].time.Day := 30, [1920].time.Hour := 13, [1920].time.Minute := 34, [1920].time.Second := 59, [1920].time.DST_ON := 1, [1921].log_data[0].min := 1.0, [1921].log_data[0].max := 1.0, [1921].log_data[0].total := 300.0, [1921].log_data[0].time := 300.0, [1921].log_data[0].minminute := 35, [1921].log_data[0].maxminute := 35, [1921].log_data[0].valid := 1, [1921].log_data[1].valid := 1, [1921].log_data[2].valid := 1, [1921].log_data[3].valid := 1, [1921].log_data[4].valid := 1, [1921].time.Year := 2022, [1921].time.Month := 4, [1921].time.Day := 30, [1921].time.Hour := 13, [1921].time.Minute := 39, [1921].time.Second := 59, [1921].time.DST_ON := 1, [1922].log_data[0].min := 1.0, [1922].log_data[0].max := 1.0, [1922].log_data[0].total := 300.0,
        [1922].log_data[0].time := 300.0, [1922].log_data[0].minminute := 40, [1922].log_data[0].maxminute := 40, [1922].log_data[0].valid := 1, [1922].log_data[1].valid := 1, [1922].log_data[2].valid := 1, [1922].log_data[3].valid := 1, [1922].log_data[4].valid := 1, [1922].time.Year := 2022, [1922].time.Month := 4, [1922].time.Day := 30, [1922].time.Hour := 13, [1922].time.Minute := 44, [1922].time.Second := 59, [1922].time.DST_ON := 1, [1923].log_data[0].min := 1.0, [1923].log_data[0].max := 1.0, [1923].log_data[0].total := 300.0, [1923].log_data[0].time := 300.0, [1923].log_data[0].minminute := 45, [1923].log_data[0].maxminute := 45, [1923].log_data[0].valid := 1, [1923].log_data[1].valid := 1, [1923].log_data[2].valid := 1, [1923].log_data[3].valid := 1, [1923].log_data[4].valid := 1, [1923].time.Year := 2022, [1923].time.Month := 4, [1923].time.Day := 30, [1923].time.Hour := 13, [1923].time.Minute := 49, [1923].time.Second := 59, [1923].time.DST_ON := 1, [1924].log_data[0].min := 1.0, [1924].log_data[0].max := 1.0, [1924].log_data[0].total := 300.0, [1924].log_data[0].time := 300.0, [1924].log_data[0].minminute := 50, [1924].log_data[0].maxminute := 50, [1924].log_data[0].valid := 1, [1924].log_data[1].valid := 1, [1924].log_data[2].valid := 1, [1924].log_data[3].valid := 1, [1924].log_data[4].valid := 1, [1924].time.Year := 2022, [1924].time.Month := 4, [1924].time.Day := 30, [1924].time.Hour := 13, [1924].time.Minute := 54, [1924].time.Second := 59, [1924].time.DST_ON := 1, [1925].log_data[0].min := 1.0, [1925].log_data[0].max := 1.0, [1925].log_data[0].total := 300.0, [1925].log_data[0].time := 300.0, [1925].log_data[0].minminute := 55, [1925].log_data[0].maxminute := 55, [1925].log_data[0].valid := 1, [1925].log_data[1].valid := 1, [1925].log_data[2].valid := 1,
        [1925].log_data[3].valid := 1, [1925].log_data[4].valid := 1, [1925].time.Year := 2022, [1925].time.Month := 4, [1925].time.Day := 30, [1925].time.Hour := 13, [1925].time.Minute := 59, [1925].time.Second := 59, [1925].time.DST_ON := 1, [1926].log_data[0].min := 1.0, [1926].log_data[0].max := 1.0, [1926].log_data[0].total := 300.0, [1926].log_data[0].time := 300.0, [1926].log_data[0].valid := 1, [1926].log_data[1].valid := 1, [1926].log_data[2].valid := 1, [1926].log_data[3].valid := 1, [1926].log_data[4].valid := 1, [1926].time.Year := 2022, [1926].time.Month := 4, [1926].time.Day := 30, [1926].time.Hour := 14, [1926].time.Minute := 4, [1926].time.Second := 59, [1926].time.DST_ON := 1, [1927].log_data[0].min := 1.0, [1927].log_data[0].max := 1.0, [1927].log_data[0].total := 300.0, [1927].log_data[0].time := 300.0, [1927].log_data[0].minminute := 5, [1927].log_data[0].maxminute := 5, [1927].log_data[0].valid := 1, [1927].log_data[1].valid := 1, [1927].log_data[2].valid := 1, [1927].log_data[3].valid := 1, [1927].log_data[4].valid := 1, [1927].time.Year := 2022, [1927].time.Month := 4, [1927].time.Day := 30, [1927].time.Hour := 14, [1927].time.Minute := 9, [1927].time.Second := 59, [1927].time.DST_ON := 1, [1928].log_data[0].min := 1.0, [1928].log_data[0].max := 1.0, [1928].log_data[0].total := 300.5, [1928].log_data[0].time := 300.5, [1928].log_data[0].minminute := 10, [1928].log_data[0].maxminute := 10, [1928].log_data[0].valid := 1, [1928].log_data[1].valid := 1, [1928].log_data[2].valid := 1, [1928].log_data[3].valid := 1, [1928].log_data[4].valid := 1, [1928].time.Year := 2022, [1928].time.Month := 4, [1928].time.Day := 30, [1928].time.Hour := 14, [1928].time.Minute := 14, [1928].time.Second := 59,
        [1928].time.DST_ON := 1, [1929].log_data[0].min := 1.0, [1929].log_data[0].max := 1.0, [1929].log_data[0].total := 300.0, [1929].log_data[0].time := 300.0, [1929].log_data[0].minminute := 15, [1929].log_data[0].maxminute := 15, [1929].log_data[0].valid := 1, [1929].log_data[1].valid := 1, [1929].log_data[2].valid := 1, [1929].log_data[3].valid := 1, [1929].log_data[4].valid := 1, [1929].time.Year := 2022, [1929].time.Month := 4, [1929].time.Day := 30, [1929].time.Hour := 14, [1929].time.Minute := 19, [1929].time.Second := 59, [1929].time.DST_ON := 1, [1930].log_data[0].min := 1.0, [1930].log_data[0].max := 1.0, [1930].log_data[0].total := 300.0, [1930].log_data[0].time := 300.0, [1930].log_data[0].minminute := 20, [1930].log_data[0].maxminute := 20, [1930].log_data[0].valid := 1, [1930].log_data[1].valid := 1, [1930].log_data[2].valid := 1, [1930].log_data[3].valid := 1, [1930].log_data[4].valid := 1, [1930].time.Year := 2022, [1930].time.Month := 4, [1930].time.Day := 30, [1930].time.Hour := 14, [1930].time.Minute := 24, [1930].time.Second := 59, [1930].time.DST_ON := 1, [1931].log_data[0].min := 1.0, [1931].log_data[0].max := 1.0, [1931].log_data[0].total := 300.0, [1931].log_data[0].time := 300.0, [1931].log_data[0].minminute := 25, [1931].log_data[0].maxminute := 25, [1931].log_data[0].valid := 1, [1931].log_data[1].valid := 1, [1931].log_data[2].valid := 1, [1931].log_data[3].valid := 1, [1931].log_data[4].valid := 1, [1931].time.Year := 2022, [1931].time.Month := 4, [1931].time.Day := 30, [1931].time.Hour := 14, [1931].time.Minute := 29, [1931].time.Second := 59, [1931].time.DST_ON := 1, [1932].log_data[0].min := 1.0, [1932].log_data[0].max := 1.0, [1932].log_data[0].total := 299.999, [1932].log_data[0].time := 299.999, [1932].log_data[0].minminute := 30,
        [1932].log_data[0].maxminute := 30, [1932].log_data[0].valid := 1, [1932].log_data[1].valid := 1, [1932].log_data[2].valid := 1, [1932].log_data[3].valid := 1, [1932].log_data[4].valid := 1, [1932].time.Year := 2022, [1932].time.Month := 4, [1932].time.Day := 30, [1932].time.Hour := 14, [1932].time.Minute := 34, [1932].time.Second := 59, [1932].time.DST_ON := 1, [1933].log_data[0].min := 1.0, [1933].log_data[0].max := 1.0, [1933].log_data[0].total := 300.0, [1933].log_data[0].time := 300.0, [1933].log_data[0].minminute := 35, [1933].log_data[0].maxminute := 35, [1933].log_data[0].valid := 1, [1933].log_data[1].valid := 1, [1933].log_data[2].valid := 1, [1933].log_data[3].valid := 1, [1933].log_data[4].valid := 1, [1933].time.Year := 2022, [1933].time.Month := 4, [1933].time.Day := 30, [1933].time.Hour := 14, [1933].time.Minute := 39, [1933].time.Second := 59, [1933].time.DST_ON := 1, [1934].log_data[0].min := 1.0, [1934].log_data[0].max := 1.0, [1934].log_data[0].total := 300.0, [1934].log_data[0].time := 300.0, [1934].log_data[0].minminute := 40, [1934].log_data[0].maxminute := 40, [1934].log_data[0].valid := 1, [1934].log_data[1].valid := 1, [1934].log_data[2].valid := 1, [1934].log_data[3].valid := 1, [1934].log_data[4].valid := 1, [1934].time.Year := 2022, [1934].time.Month := 4, [1934].time.Day := 30, [1934].time.Hour := 14, [1934].time.Minute := 44, [1934].time.Second := 59, [1934].time.DST_ON := 1, [1935].log_data[0].min := 1.0, [1935].log_data[0].max := 1.0, [1935].log_data[0].total := 300.0, [1935].log_data[0].time := 300.0, [1935].log_data[0].minminute := 45, [1935].log_data[0].maxminute := 45, [1935].log_data[0].valid := 1, [1935].log_data[1].valid := 1, [1935].log_data[2].valid := 1, [1935].log_data[3].valid := 1, [1935].log_data[4].valid := 1,
        [1935].time.Year := 2022, [1935].time.Month := 4, [1935].time.Day := 30, [1935].time.Hour := 14, [1935].time.Minute := 49, [1935].time.Second := 59, [1935].time.DST_ON := 1, [1936].log_data[0].min := 1.0, [1936].log_data[0].max := 1.0, [1936].log_data[0].total := 300.0, [1936].log_data[0].time := 300.0, [1936].log_data[0].minminute := 50, [1936].log_data[0].maxminute := 50, [1936].log_data[0].valid := 1, [1936].log_data[1].valid := 1, [1936].log_data[2].valid := 1, [1936].log_data[3].valid := 1, [1936].log_data[4].valid := 1, [1936].time.Year := 2022, [1936].time.Month := 4, [1936].time.Day := 30, [1936].time.Hour := 14, [1936].time.Minute := 54, [1936].time.Second := 59, [1936].time.DST_ON := 1, [1937].log_data[0].min := 1.0, [1937].log_data[0].max := 1.0, [1937].log_data[0].total := 300.0, [1937].log_data[0].time := 300.0, [1937].log_data[0].minminute := 55, [1937].log_data[0].maxminute := 55, [1937].log_data[0].valid := 1, [1937].log_data[1].valid := 1, [1937].log_data[2].valid := 1, [1937].log_data[3].valid := 1, [1937].log_data[4].valid := 1, [1937].time.Year := 2022, [1937].time.Month := 4, [1937].time.Day := 30, [1937].time.Hour := 14, [1937].time.Minute := 59, [1937].time.Second := 59, [1937].time.DST_ON := 1, [1938].log_data[0].min := 1.0, [1938].log_data[0].max := 1.0, [1938].log_data[0].total := 300.0, [1938].log_data[0].time := 300.0, [1938].log_data[0].valid := 1, [1938].log_data[1].valid := 1, [1938].log_data[2].valid := 1, [1938].log_data[3].valid := 1, [1938].log_data[4].valid := 1, [1938].time.Year := 2022, [1938].time.Month := 4, [1938].time.Day := 30, [1938].time.Hour := 15, [1938].time.Minute := 4, [1938].time.Second := 59, [1938].time.DST_ON := 1, [1939].log_data[0].min := 1.0,
        [1939].log_data[0].max := 1.0, [1939].log_data[0].total := 300.0, [1939].log_data[0].time := 300.0, [1939].log_data[0].minminute := 5, [1939].log_data[0].maxminute := 5, [1939].log_data[0].valid := 1, [1939].log_data[1].valid := 1, [1939].log_data[2].valid := 1, [1939].log_data[3].valid := 1, [1939].log_data[4].valid := 1, [1939].time.Year := 2022, [1939].time.Month := 4, [1939].time.Day := 30, [1939].time.Hour := 15, [1939].time.Minute := 9, [1939].time.Second := 59, [1939].time.DST_ON := 1, [1940].log_data[0].min := 1.0, [1940].log_data[0].max := 1.0, [1940].log_data[0].total := 300.0, [1940].log_data[0].time := 300.0, [1940].log_data[0].minminute := 10, [1940].log_data[0].maxminute := 10, [1940].log_data[0].valid := 1, [1940].log_data[1].valid := 1, [1940].log_data[2].valid := 1, [1940].log_data[3].valid := 1, [1940].log_data[4].valid := 1, [1940].time.Year := 2022, [1940].time.Month := 4, [1940].time.Day := 30, [1940].time.Hour := 15, [1940].time.Minute := 14, [1940].time.Second := 59, [1940].time.DST_ON := 1, [1941].log_data[0].min := 1.0, [1941].log_data[0].max := 1.0, [1941].log_data[0].total := 300.0, [1941].log_data[0].time := 300.0, [1941].log_data[0].minminute := 15, [1941].log_data[0].maxminute := 15, [1941].log_data[0].valid := 1, [1941].log_data[1].valid := 1, [1941].log_data[2].valid := 1, [1941].log_data[3].valid := 1, [1941].log_data[4].valid := 1, [1941].time.Year := 2022, [1941].time.Month := 4, [1941].time.Day := 30, [1941].time.Hour := 15, [1941].time.Minute := 19, [1941].time.Second := 59, [1941].time.DST_ON := 1, [1942].log_data[0].min := 1.0, [1942].log_data[0].max := 1.0, [1942].log_data[0].total := 300.0, [1942].log_data[0].time := 300.0, [1942].log_data[0].minminute := 20, [1942].log_data[0].maxminute := 20, [1942].log_data[0].valid := 1,
        [1942].log_data[1].valid := 1, [1942].log_data[2].valid := 1, [1942].log_data[3].valid := 1, [1942].log_data[4].valid := 1, [1942].time.Year := 2022, [1942].time.Month := 4, [1942].time.Day := 30, [1942].time.Hour := 15, [1942].time.Minute := 24, [1942].time.Second := 59, [1942].time.DST_ON := 1, [1943].log_data[0].min := 1.0, [1943].log_data[0].max := 1.0, [1943].log_data[0].total := 300.0, [1943].log_data[0].time := 300.0, [1943].log_data[0].minminute := 25, [1943].log_data[0].maxminute := 25, [1943].log_data[0].valid := 1, [1943].log_data[1].valid := 1, [1943].log_data[2].valid := 1, [1943].log_data[3].valid := 1, [1943].log_data[4].valid := 1, [1943].time.Year := 2022, [1943].time.Month := 4, [1943].time.Day := 30, [1943].time.Hour := 15, [1943].time.Minute := 29, [1943].time.Second := 59, [1943].time.DST_ON := 1, [1944].log_data[0].min := 1.0, [1944].log_data[0].max := 1.0, [1944].log_data[0].total := 300.0, [1944].log_data[0].time := 300.0, [1944].log_data[0].minminute := 30, [1944].log_data[0].maxminute := 30, [1944].log_data[0].valid := 1, [1944].log_data[1].valid := 1, [1944].log_data[2].valid := 1, [1944].log_data[3].valid := 1, [1944].log_data[4].valid := 1, [1944].time.Year := 2022, [1944].time.Month := 4, [1944].time.Day := 30, [1944].time.Hour := 15, [1944].time.Minute := 34, [1944].time.Second := 59, [1944].time.DST_ON := 1, [1945].log_data[0].min := 1.0, [1945].log_data[0].max := 1.0, [1945].log_data[0].total := 300.0, [1945].log_data[0].time := 300.0, [1945].log_data[0].minminute := 35, [1945].log_data[0].maxminute := 35, [1945].log_data[0].valid := 1, [1945].log_data[1].valid := 1, [1945].log_data[2].valid := 1, [1945].log_data[3].valid := 1, [1945].log_data[4].valid := 1, [1945].time.Year := 2022, [1945].time.Month := 4,
        [1945].time.Day := 30, [1945].time.Hour := 15, [1945].time.Minute := 39, [1945].time.Second := 59, [1945].time.DST_ON := 1, [1946].log_data[0].min := 1.0, [1946].log_data[0].max := 1.0, [1946].log_data[0].total := 300.0, [1946].log_data[0].time := 300.0, [1946].log_data[0].minminute := 40, [1946].log_data[0].maxminute := 40, [1946].log_data[0].valid := 1, [1946].log_data[1].valid := 1, [1946].log_data[2].valid := 1, [1946].log_data[3].valid := 1, [1946].log_data[4].valid := 1, [1946].time.Year := 2022, [1946].time.Month := 4, [1946].time.Day := 30, [1946].time.Hour := 15, [1946].time.Minute := 44, [1946].time.Second := 59, [1946].time.DST_ON := 1, [1947].log_data[0].min := 1.0, [1947].log_data[0].max := 1.0, [1947].log_data[0].total := 300.0, [1947].log_data[0].time := 300.0, [1947].log_data[0].minminute := 45, [1947].log_data[0].maxminute := 45, [1947].log_data[0].valid := 1, [1947].log_data[1].valid := 1, [1947].log_data[2].valid := 1, [1947].log_data[3].valid := 1, [1947].log_data[4].valid := 1, [1947].time.Year := 2022, [1947].time.Month := 4, [1947].time.Day := 30, [1947].time.Hour := 15, [1947].time.Minute := 49, [1947].time.Second := 59, [1947].time.DST_ON := 1, [1948].log_data[0].min := 1.0, [1948].log_data[0].max := 1.0, [1948].log_data[0].total := 300.0, [1948].log_data[0].time := 300.0, [1948].log_data[0].minminute := 50, [1948].log_data[0].maxminute := 50, [1948].log_data[0].valid := 1, [1948].log_data[1].valid := 1, [1948].log_data[2].valid := 1, [1948].log_data[3].valid := 1, [1948].log_data[4].valid := 1, [1948].time.Year := 2022, [1948].time.Month := 4, [1948].time.Day := 30, [1948].time.Hour := 15, [1948].time.Minute := 54, [1948].time.Second := 59, [1948].time.DST_ON := 1, [1949].log_data[0].min := 1.0,
        [1949].log_data[0].max := 1.0, [1949].log_data[0].total := 300.0, [1949].log_data[0].time := 300.0, [1949].log_data[0].minminute := 55, [1949].log_data[0].maxminute := 55, [1949].log_data[0].valid := 1, [1949].log_data[1].valid := 1, [1949].log_data[2].valid := 1, [1949].log_data[3].valid := 1, [1949].log_data[4].valid := 1, [1949].time.Year := 2022, [1949].time.Month := 4, [1949].time.Day := 30, [1949].time.Hour := 15, [1949].time.Minute := 59, [1949].time.Second := 59, [1949].time.DST_ON := 1, [1950].log_data[0].min := 1.0, [1950].log_data[0].max := 1.0, [1950].log_data[0].total := 300.0, [1950].log_data[0].time := 300.0, [1950].log_data[0].valid := 1, [1950].log_data[1].valid := 1, [1950].log_data[2].valid := 1, [1950].log_data[3].valid := 1, [1950].log_data[4].valid := 1, [1950].time.Year := 2022, [1950].time.Month := 4, [1950].time.Day := 30, [1950].time.Hour := 16, [1950].time.Minute := 4, [1950].time.Second := 59, [1950].time.DST_ON := 1, [1951].log_data[0].min := 1.0, [1951].log_data[0].max := 1.0, [1951].log_data[0].total := 300.0, [1951].log_data[0].time := 300.0, [1951].log_data[0].minminute := 5, [1951].log_data[0].maxminute := 5, [1951].log_data[0].valid := 1, [1951].log_data[1].valid := 1, [1951].log_data[2].valid := 1, [1951].log_data[3].valid := 1, [1951].log_data[4].valid := 1, [1951].time.Year := 2022, [1951].time.Month := 4, [1951].time.Day := 30, [1951].time.Hour := 16, [1951].time.Minute := 9, [1951].time.Second := 59, [1951].time.DST_ON := 1, [1952].log_data[0].min := 1.0, [1952].log_data[0].max := 1.0, [1952].log_data[0].total := 300.0, [1952].log_data[0].time := 300.0, [1952].log_data[0].minminute := 10, [1952].log_data[0].maxminute := 10, [1952].log_data[0].valid := 1, [1952].log_data[1].valid := 1, [1952].log_data[2].valid := 1,
        [1952].log_data[3].valid := 1, [1952].log_data[4].valid := 1, [1952].time.Year := 2022, [1952].time.Month := 4, [1952].time.Day := 30, [1952].time.Hour := 16, [1952].time.Minute := 14, [1952].time.Second := 59, [1952].time.DST_ON := 1, [1953].log_data[0].min := 1.0, [1953].log_data[0].max := 1.0, [1953].log_data[0].total := 300.0, [1953].log_data[0].time := 300.0, [1953].log_data[0].minminute := 15, [1953].log_data[0].maxminute := 15, [1953].log_data[0].valid := 1, [1953].log_data[1].valid := 1, [1953].log_data[2].valid := 1, [1953].log_data[3].valid := 1, [1953].log_data[4].valid := 1, [1953].time.Year := 2022, [1953].time.Month := 4, [1953].time.Day := 30, [1953].time.Hour := 16, [1953].time.Minute := 19, [1953].time.Second := 59, [1953].time.DST_ON := 1, [1954].log_data[0].min := 1.0, [1954].log_data[0].max := 1.0, [1954].log_data[0].total := 300.0, [1954].log_data[0].time := 300.0, [1954].log_data[0].minminute := 20, [1954].log_data[0].maxminute := 20, [1954].log_data[0].valid := 1, [1954].log_data[1].valid := 1, [1954].log_data[2].valid := 1, [1954].log_data[3].valid := 1, [1954].log_data[4].valid := 1, [1954].time.Year := 2022, [1954].time.Month := 4, [1954].time.Day := 30, [1954].time.Hour := 16, [1954].time.Minute := 24, [1954].time.Second := 59, [1954].time.DST_ON := 1, [1955].log_data[0].min := 1.0, [1955].log_data[0].max := 1.0, [1955].log_data[0].total := 300.0, [1955].log_data[0].time := 300.0, [1955].log_data[0].minminute := 25, [1955].log_data[0].maxminute := 25, [1955].log_data[0].valid := 1, [1955].log_data[1].valid := 1, [1955].log_data[2].valid := 1, [1955].log_data[3].valid := 1, [1955].log_data[4].valid := 1, [1955].time.Year := 2022, [1955].time.Month := 4, [1955].time.Day := 30, [1955].time.Hour := 16,
        [1955].time.Minute := 29, [1955].time.Second := 59, [1955].time.DST_ON := 1, [1956].log_data[0].min := 1.0, [1956].log_data[0].max := 1.0, [1956].log_data[0].total := 299.999, [1956].log_data[0].time := 299.999, [1956].log_data[0].minminute := 30, [1956].log_data[0].maxminute := 30, [1956].log_data[0].valid := 1, [1956].log_data[1].valid := 1, [1956].log_data[2].valid := 1, [1956].log_data[3].valid := 1, [1956].log_data[4].valid := 1, [1956].time.Year := 2022, [1956].time.Month := 4, [1956].time.Day := 30, [1956].time.Hour := 16, [1956].time.Minute := 34, [1956].time.Second := 59, [1956].time.DST_ON := 1, [1957].log_data[0].min := 1.0, [1957].log_data[0].max := 1.0, [1957].log_data[0].total := 300.0, [1957].log_data[0].time := 300.0, [1957].log_data[0].minminute := 35, [1957].log_data[0].maxminute := 35, [1957].log_data[0].valid := 1, [1957].log_data[1].valid := 1, [1957].log_data[2].valid := 1, [1957].log_data[3].valid := 1, [1957].log_data[4].valid := 1, [1957].time.Year := 2022, [1957].time.Month := 4, [1957].time.Day := 30, [1957].time.Hour := 16, [1957].time.Minute := 39, [1957].time.Second := 59, [1957].time.DST_ON := 1, [1958].log_data[0].min := 1.0, [1958].log_data[0].max := 1.0, [1958].log_data[0].total := 300.0, [1958].log_data[0].time := 300.0, [1958].log_data[0].minminute := 40, [1958].log_data[0].maxminute := 40, [1958].log_data[0].valid := 1, [1958].log_data[1].valid := 1, [1958].log_data[2].valid := 1, [1958].log_data[3].valid := 1, [1958].log_data[4].valid := 1, [1958].time.Year := 2022, [1958].time.Month := 4, [1958].time.Day := 30, [1958].time.Hour := 16, [1958].time.Minute := 44, [1958].time.Second := 59, [1958].time.DST_ON := 1, [1959].log_data[0].min := 1.0, [1959].log_data[0].max := 1.0, [1959].log_data[0].total := 300.0,
        [1959].log_data[0].time := 300.0, [1959].log_data[0].minminute := 45, [1959].log_data[0].maxminute := 45, [1959].log_data[0].valid := 1, [1959].log_data[1].valid := 1, [1959].log_data[2].valid := 1, [1959].log_data[3].valid := 1, [1959].log_data[4].valid := 1, [1959].time.Year := 2022, [1959].time.Month := 4, [1959].time.Day := 30, [1959].time.Hour := 16, [1959].time.Minute := 49, [1959].time.Second := 59, [1959].time.DST_ON := 1, [1960].log_data[0].min := 1.0, [1960].log_data[0].max := 1.0, [1960].log_data[0].total := 300.0, [1960].log_data[0].time := 300.0, [1960].log_data[0].minminute := 50, [1960].log_data[0].maxminute := 50, [1960].log_data[0].valid := 1, [1960].log_data[1].valid := 1, [1960].log_data[2].valid := 1, [1960].log_data[3].valid := 1, [1960].log_data[4].valid := 1, [1960].time.Year := 2022, [1960].time.Month := 4, [1960].time.Day := 30, [1960].time.Hour := 16, [1960].time.Minute := 54, [1960].time.Second := 59, [1960].time.DST_ON := 1, [1961].log_data[0].min := 1.0, [1961].log_data[0].max := 1.0, [1961].log_data[0].total := 300.0, [1961].log_data[0].time := 300.0, [1961].log_data[0].minminute := 55, [1961].log_data[0].maxminute := 55, [1961].log_data[0].valid := 1, [1961].log_data[1].valid := 1, [1961].log_data[2].valid := 1, [1961].log_data[3].valid := 1, [1961].log_data[4].valid := 1, [1961].time.Year := 2022, [1961].time.Month := 4, [1961].time.Day := 30, [1961].time.Hour := 16, [1961].time.Minute := 59, [1961].time.Second := 59, [1961].time.DST_ON := 1, [1962].log_data[0].min := 1.0, [1962].log_data[0].max := 1.0, [1962].log_data[0].total := 300.0, [1962].log_data[0].time := 300.0, [1962].log_data[0].valid := 1, [1962].log_data[1].valid := 1, [1962].log_data[2].valid := 1, [1962].log_data[3].valid := 1, [1962].log_data[4].valid := 1,
        [1962].time.Year := 2022, [1962].time.Month := 4, [1962].time.Day := 30, [1962].time.Hour := 17, [1962].time.Minute := 4, [1962].time.Second := 59, [1962].time.DST_ON := 1, [1963].log_data[0].min := 1.0, [1963].log_data[0].max := 1.0, [1963].log_data[0].total := 300.0, [1963].log_data[0].time := 300.0, [1963].log_data[0].minminute := 5, [1963].log_data[0].maxminute := 5, [1963].log_data[0].valid := 1, [1963].log_data[1].valid := 1, [1963].log_data[2].valid := 1, [1963].log_data[3].valid := 1, [1963].log_data[4].valid := 1, [1963].time.Year := 2022, [1963].time.Month := 4, [1963].time.Day := 30, [1963].time.Hour := 17, [1963].time.Minute := 9, [1963].time.Second := 59, [1963].time.DST_ON := 1, [1964].log_data[0].min := 1.0, [1964].log_data[0].max := 1.0, [1964].log_data[0].total := 300.0, [1964].log_data[0].time := 300.0, [1964].log_data[0].minminute := 10, [1964].log_data[0].maxminute := 10, [1964].log_data[0].valid := 1, [1964].log_data[1].valid := 1, [1964].log_data[2].valid := 1, [1964].log_data[3].valid := 1, [1964].log_data[4].valid := 1, [1964].time.Year := 2022, [1964].time.Month := 4, [1964].time.Day := 30, [1964].time.Hour := 17, [1964].time.Minute := 14, [1964].time.Second := 59, [1964].time.DST_ON := 1, [1965].log_data[0].min := 1.0, [1965].log_data[0].max := 1.0, [1965].log_data[0].total := 300.0, [1965].log_data[0].time := 300.0, [1965].log_data[0].minminute := 15, [1965].log_data[0].maxminute := 15, [1965].log_data[0].valid := 1, [1965].log_data[1].valid := 1, [1965].log_data[2].valid := 1, [1965].log_data[3].valid := 1, [1965].log_data[4].valid := 1, [1965].time.Year := 2022, [1965].time.Month := 4, [1965].time.Day := 30, [1965].time.Hour := 17, [1965].time.Minute := 19, [1965].time.Second := 59,
        [1965].time.DST_ON := 1, [1966].log_data[0].min := 1.0, [1966].log_data[0].max := 1.0, [1966].log_data[0].total := 300.0, [1966].log_data[0].time := 300.0, [1966].log_data[0].minminute := 20, [1966].log_data[0].maxminute := 20, [1966].log_data[0].valid := 1, [1966].log_data[1].valid := 1, [1966].log_data[2].valid := 1, [1966].log_data[3].valid := 1, [1966].log_data[4].valid := 1, [1966].time.Year := 2022, [1966].time.Month := 4, [1966].time.Day := 30, [1966].time.Hour := 17, [1966].time.Minute := 24, [1966].time.Second := 59, [1966].time.DST_ON := 1, [1967].log_data[0].min := 1.0, [1967].log_data[0].max := 1.0, [1967].log_data[0].total := 300.0, [1967].log_data[0].time := 300.0, [1967].log_data[0].minminute := 25, [1967].log_data[0].maxminute := 25, [1967].log_data[0].valid := 1, [1967].log_data[1].valid := 1, [1967].log_data[2].valid := 1, [1967].log_data[3].valid := 1, [1967].log_data[4].valid := 1, [1967].time.Year := 2022, [1967].time.Month := 4, [1967].time.Day := 30, [1967].time.Hour := 17, [1967].time.Minute := 29, [1967].time.Second := 59, [1967].time.DST_ON := 1, [1968].log_data[0].min := 1.0, [1968].log_data[0].max := 1.0, [1968].log_data[0].total := 300.0, [1968].log_data[0].time := 300.0, [1968].log_data[0].minminute := 30, [1968].log_data[0].maxminute := 30, [1968].log_data[0].valid := 1, [1968].log_data[1].valid := 1, [1968].log_data[2].valid := 1, [1968].log_data[3].valid := 1, [1968].log_data[4].valid := 1, [1968].time.Year := 2022, [1968].time.Month := 4, [1968].time.Day := 30, [1968].time.Hour := 17, [1968].time.Minute := 34, [1968].time.Second := 59, [1968].time.DST_ON := 1, [1969].log_data[0].min := 1.0, [1969].log_data[0].max := 1.0, [1969].log_data[0].total := 300.0, [1969].log_data[0].time := 300.0, [1969].log_data[0].minminute := 35,
        [1969].log_data[0].maxminute := 35, [1969].log_data[0].valid := 1, [1969].log_data[1].valid := 1, [1969].log_data[2].valid := 1, [1969].log_data[3].valid := 1, [1969].log_data[4].valid := 1, [1969].time.Year := 2022, [1969].time.Month := 4, [1969].time.Day := 30, [1969].time.Hour := 17, [1969].time.Minute := 39, [1969].time.Second := 59, [1969].time.DST_ON := 1, [1970].log_data[0].min := 1.0, [1970].log_data[0].max := 1.0, [1970].log_data[0].total := 300.0, [1970].log_data[0].time := 300.0, [1970].log_data[0].minminute := 40, [1970].log_data[0].maxminute := 40, [1970].log_data[0].valid := 1, [1970].log_data[1].valid := 1, [1970].log_data[2].valid := 1, [1970].log_data[3].valid := 1, [1970].log_data[4].valid := 1, [1970].time.Year := 2022, [1970].time.Month := 4, [1970].time.Day := 30, [1970].time.Hour := 17, [1970].time.Minute := 44, [1970].time.Second := 59, [1970].time.DST_ON := 1, [1971].log_data[0].min := 1.0, [1971].log_data[0].max := 1.0, [1971].log_data[0].total := 300.0, [1971].log_data[0].time := 300.0, [1971].log_data[0].minminute := 45, [1971].log_data[0].maxminute := 45, [1971].log_data[0].valid := 1, [1971].log_data[1].valid := 1, [1971].log_data[2].valid := 1, [1971].log_data[3].valid := 1, [1971].log_data[4].valid := 1, [1971].time.Year := 2022, [1971].time.Month := 4, [1971].time.Day := 30, [1971].time.Hour := 17, [1971].time.Minute := 49, [1971].time.Second := 59, [1971].time.DST_ON := 1, [1972].log_data[0].min := 1.0, [1972].log_data[0].max := 1.0, [1972].log_data[0].total := 300.0, [1972].log_data[0].time := 300.0, [1972].log_data[0].minminute := 50, [1972].log_data[0].maxminute := 50, [1972].log_data[0].valid := 1, [1972].log_data[1].valid := 1, [1972].log_data[2].valid := 1, [1972].log_data[3].valid := 1, [1972].log_data[4].valid := 1,
        [1972].time.Year := 2022, [1972].time.Month := 4, [1972].time.Day := 30, [1972].time.Hour := 17, [1972].time.Minute := 54, [1972].time.Second := 59, [1972].time.DST_ON := 1, [1973].log_data[0].min := 1.0, [1973].log_data[0].max := 1.0, [1973].log_data[0].total := 300.0, [1973].log_data[0].time := 300.0, [1973].log_data[0].minminute := 55, [1973].log_data[0].maxminute := 55, [1973].log_data[0].valid := 1, [1973].log_data[1].valid := 1, [1973].log_data[2].valid := 1, [1973].log_data[3].valid := 1, [1973].log_data[4].valid := 1, [1973].time.Year := 2022, [1973].time.Month := 4, [1973].time.Day := 30, [1973].time.Hour := 17, [1973].time.Minute := 59, [1973].time.Second := 59, [1973].time.DST_ON := 1, [1974].log_data[0].min := 1.0, [1974].log_data[0].max := 1.0, [1974].log_data[0].total := 300.0, [1974].log_data[0].time := 300.0, [1974].log_data[0].valid := 1, [1974].log_data[1].valid := 1, [1974].log_data[2].valid := 1, [1974].log_data[3].valid := 1, [1974].log_data[4].valid := 1, [1974].time.Year := 2022, [1974].time.Month := 4, [1974].time.Day := 30, [1974].time.Hour := 18, [1974].time.Minute := 4, [1974].time.Second := 59, [1974].time.DST_ON := 1, [1975].log_data[0].min := 1.0, [1975].log_data[0].max := 1.0, [1975].log_data[0].total := 300.0, [1975].log_data[0].time := 300.0, [1975].log_data[0].minminute := 5, [1975].log_data[0].maxminute := 5, [1975].log_data[0].valid := 1, [1975].log_data[1].valid := 1, [1975].log_data[2].valid := 1, [1975].log_data[3].valid := 1, [1975].log_data[4].valid := 1, [1975].time.Year := 2022, [1975].time.Month := 4, [1975].time.Day := 30, [1975].time.Hour := 18, [1975].time.Minute := 9, [1975].time.Second := 59, [1975].time.DST_ON := 1, [1976].log_data[0].min := 1.0,
        [1976].log_data[0].max := 1.0, [1976].log_data[0].total := 300.0, [1976].log_data[0].time := 300.0, [1976].log_data[0].minminute := 10, [1976].log_data[0].maxminute := 10, [1976].log_data[0].valid := 1, [1976].log_data[1].valid := 1, [1976].log_data[2].valid := 1, [1976].log_data[3].valid := 1, [1976].log_data[4].valid := 1, [1976].time.Year := 2022, [1976].time.Month := 4, [1976].time.Day := 30, [1976].time.Hour := 18, [1976].time.Minute := 14, [1976].time.Second := 59, [1976].time.DST_ON := 1, [1977].log_data[0].min := 1.0, [1977].log_data[0].max := 1.0, [1977].log_data[0].total := 300.0, [1977].log_data[0].time := 300.0, [1977].log_data[0].minminute := 15, [1977].log_data[0].maxminute := 15, [1977].log_data[0].valid := 1, [1977].log_data[1].valid := 1, [1977].log_data[2].valid := 1, [1977].log_data[3].valid := 1, [1977].log_data[4].valid := 1, [1977].time.Year := 2022, [1977].time.Month := 4, [1977].time.Day := 30, [1977].time.Hour := 18, [1977].time.Minute := 19, [1977].time.Second := 59, [1977].time.DST_ON := 1, [1978].log_data[0].min := 1.0, [1978].log_data[0].max := 1.0, [1978].log_data[0].total := 300.0, [1978].log_data[0].time := 300.0, [1978].log_data[0].minminute := 20, [1978].log_data[0].maxminute := 20, [1978].log_data[0].valid := 1, [1978].log_data[1].valid := 1, [1978].log_data[2].valid := 1, [1978].log_data[3].valid := 1, [1978].log_data[4].valid := 1, [1978].time.Year := 2022, [1978].time.Month := 4, [1978].time.Day := 30, [1978].time.Hour := 18, [1978].time.Minute := 24, [1978].time.Second := 59, [1978].time.DST_ON := 1, [1979].log_data[0].min := 1.0, [1979].log_data[0].max := 1.0, [1979].log_data[0].total := 300.0, [1979].log_data[0].time := 300.0, [1979].log_data[0].minminute := 25, [1979].log_data[0].maxminute := 25, [1979].log_data[0].valid := 1,
        [1979].log_data[1].valid := 1, [1979].log_data[2].valid := 1, [1979].log_data[3].valid := 1, [1979].log_data[4].valid := 1, [1979].time.Year := 2022, [1979].time.Month := 4, [1979].time.Day := 30, [1979].time.Hour := 18, [1979].time.Minute := 29, [1979].time.Second := 59, [1979].time.DST_ON := 1, [1980].log_data[0].min := 1.0, [1980].log_data[0].max := 1.0, [1980].log_data[0].total := 300.0, [1980].log_data[0].time := 300.0, [1980].log_data[0].minminute := 30, [1980].log_data[0].maxminute := 30, [1980].log_data[0].valid := 1, [1980].log_data[1].valid := 1, [1980].log_data[2].valid := 1, [1980].log_data[3].valid := 1, [1980].log_data[4].valid := 1, [1980].time.Year := 2022, [1980].time.Month := 4, [1980].time.Day := 30, [1980].time.Hour := 18, [1980].time.Minute := 34, [1980].time.Second := 59, [1980].time.DST_ON := 1, [1981].log_data[0].min := 1.0, [1981].log_data[0].max := 1.0, [1981].log_data[0].total := 300.0, [1981].log_data[0].time := 300.0, [1981].log_data[0].minminute := 35, [1981].log_data[0].maxminute := 35, [1981].log_data[0].valid := 1, [1981].log_data[1].valid := 1, [1981].log_data[2].valid := 1, [1981].log_data[3].valid := 1, [1981].log_data[4].valid := 1, [1981].time.Year := 2022, [1981].time.Month := 4, [1981].time.Day := 30, [1981].time.Hour := 18, [1981].time.Minute := 39, [1981].time.Second := 59, [1981].time.DST_ON := 1, [1982].log_data[0].min := 1.0, [1982].log_data[0].max := 1.0, [1982].log_data[0].total := 300.0, [1982].log_data[0].time := 300.0, [1982].log_data[0].minminute := 40, [1982].log_data[0].maxminute := 40, [1982].log_data[0].valid := 1, [1982].log_data[1].valid := 1, [1982].log_data[2].valid := 1, [1982].log_data[3].valid := 1, [1982].log_data[4].valid := 1, [1982].time.Year := 2022, [1982].time.Month := 4,
        [1982].time.Day := 30, [1982].time.Hour := 18, [1982].time.Minute := 44, [1982].time.Second := 59, [1982].time.DST_ON := 1, [1983].log_data[0].min := 1.0, [1983].log_data[0].max := 1.0, [1983].log_data[0].total := 300.0, [1983].log_data[0].time := 300.0, [1983].log_data[0].minminute := 45, [1983].log_data[0].maxminute := 45, [1983].log_data[0].valid := 1, [1983].log_data[1].valid := 1, [1983].log_data[2].valid := 1, [1983].log_data[3].valid := 1, [1983].log_data[4].valid := 1, [1983].time.Year := 2022, [1983].time.Month := 4, [1983].time.Day := 30, [1983].time.Hour := 18, [1983].time.Minute := 49, [1983].time.Second := 59, [1983].time.DST_ON := 1, [1984].log_data[0].min := 1.0, [1984].log_data[0].max := 1.0, [1984].log_data[0].total := 300.0, [1984].log_data[0].time := 300.0, [1984].log_data[0].minminute := 50, [1984].log_data[0].maxminute := 50, [1984].log_data[0].valid := 1, [1984].log_data[1].valid := 1, [1984].log_data[2].valid := 1, [1984].log_data[3].valid := 1, [1984].log_data[4].valid := 1, [1984].time.Year := 2022, [1984].time.Month := 4, [1984].time.Day := 30, [1984].time.Hour := 18, [1984].time.Minute := 54, [1984].time.Second := 59, [1984].time.DST_ON := 1, [1985].log_data[0].min := 1.0, [1985].log_data[0].max := 1.0, [1985].log_data[0].total := 300.0, [1985].log_data[0].time := 300.0, [1985].log_data[0].minminute := 55, [1985].log_data[0].maxminute := 55, [1985].log_data[0].valid := 1, [1985].log_data[1].valid := 1, [1985].log_data[2].valid := 1, [1985].log_data[3].valid := 1, [1985].log_data[4].valid := 1, [1985].time.Year := 2022, [1985].time.Month := 4, [1985].time.Day := 30, [1985].time.Hour := 18, [1985].time.Minute := 59, [1985].time.Second := 59, [1985].time.DST_ON := 1, [1986].log_data[0].min := 1.0,
        [1986].log_data[0].max := 1.0, [1986].log_data[0].total := 299.999, [1986].log_data[0].time := 299.999, [1986].log_data[0].valid := 1, [1986].log_data[1].valid := 1, [1986].log_data[2].valid := 1, [1986].log_data[3].valid := 1, [1986].log_data[4].valid := 1, [1986].time.Year := 2022, [1986].time.Month := 4, [1986].time.Day := 30, [1986].time.Hour := 19, [1986].time.Minute := 4, [1986].time.Second := 59, [1986].time.DST_ON := 1, [1987].log_data[0].min := 1.0, [1987].log_data[0].max := 1.0, [1987].log_data[0].total := 300.0, [1987].log_data[0].time := 300.0, [1987].log_data[0].minminute := 5, [1987].log_data[0].maxminute := 5, [1987].log_data[0].valid := 1, [1987].log_data[1].valid := 1, [1987].log_data[2].valid := 1, [1987].log_data[3].valid := 1, [1987].log_data[4].valid := 1, [1987].time.Year := 2022, [1987].time.Month := 4, [1987].time.Day := 30, [1987].time.Hour := 19, [1987].time.Minute := 9, [1987].time.Second := 59, [1987].time.DST_ON := 1, [1988].log_data[0].min := 1.0, [1988].log_data[0].max := 1.0, [1988].log_data[0].total := 300.0, [1988].log_data[0].time := 300.0, [1988].log_data[0].minminute := 10, [1988].log_data[0].maxminute := 10, [1988].log_data[0].valid := 1, [1988].log_data[1].valid := 1, [1988].log_data[2].valid := 1, [1988].log_data[3].valid := 1, [1988].log_data[4].valid := 1, [1988].time.Year := 2022, [1988].time.Month := 4, [1988].time.Day := 30, [1988].time.Hour := 19, [1988].time.Minute := 14, [1988].time.Second := 59, [1988].time.DST_ON := 1, [1989].log_data[0].min := 1.0, [1989].log_data[0].max := 1.0, [1989].log_data[0].total := 300.0, [1989].log_data[0].time := 300.0, [1989].log_data[0].minminute := 15, [1989].log_data[0].maxminute := 15, [1989].log_data[0].valid := 1, [1989].log_data[1].valid := 1, [1989].log_data[2].valid := 1,
        [1989].log_data[3].valid := 1, [1989].log_data[4].valid := 1, [1989].time.Year := 2022, [1989].time.Month := 4, [1989].time.Day := 30, [1989].time.Hour := 19, [1989].time.Minute := 19, [1989].time.Second := 59, [1989].time.DST_ON := 1, [1990].log_data[0].min := 1.0, [1990].log_data[0].max := 1.0, [1990].log_data[0].total := 300.0, [1990].log_data[0].time := 300.0, [1990].log_data[0].minminute := 20, [1990].log_data[0].maxminute := 20, [1990].log_data[0].valid := 1, [1990].log_data[1].valid := 1, [1990].log_data[2].valid := 1, [1990].log_data[3].valid := 1, [1990].log_data[4].valid := 1, [1990].time.Year := 2022, [1990].time.Month := 4, [1990].time.Day := 30, [1990].time.Hour := 19, [1990].time.Minute := 24, [1990].time.Second := 59, [1990].time.DST_ON := 1, [1991].log_data[0].min := 1.0, [1991].log_data[0].max := 1.0, [1991].log_data[0].total := 300.0, [1991].log_data[0].time := 300.0, [1991].log_data[0].minminute := 25, [1991].log_data[0].maxminute := 25, [1991].log_data[0].valid := 1, [1991].log_data[1].valid := 1, [1991].log_data[2].valid := 1, [1991].log_data[3].valid := 1, [1991].log_data[4].valid := 1, [1991].time.Year := 2022, [1991].time.Month := 4, [1991].time.Day := 30, [1991].time.Hour := 19, [1991].time.Minute := 29, [1991].time.Second := 59, [1991].time.DST_ON := 1, [1992].log_data[0].min := 1.0, [1992].log_data[0].max := 1.0, [1992].log_data[0].total := 300.0, [1992].log_data[0].time := 300.0, [1992].log_data[0].minminute := 30, [1992].log_data[0].maxminute := 30, [1992].log_data[0].valid := 1, [1992].log_data[1].valid := 1, [1992].log_data[2].valid := 1, [1992].log_data[3].valid := 1, [1992].log_data[4].valid := 1, [1992].time.Year := 2022, [1992].time.Month := 4, [1992].time.Day := 30, [1992].time.Hour := 19,
        [1992].time.Minute := 34, [1992].time.Second := 59, [1992].time.DST_ON := 1, [1993].log_data[0].min := 1.0, [1993].log_data[0].max := 1.0, [1993].log_data[0].total := 300.0, [1993].log_data[0].time := 300.0, [1993].log_data[0].minminute := 35, [1993].log_data[0].maxminute := 35, [1993].log_data[0].valid := 1, [1993].log_data[1].valid := 1, [1993].log_data[2].valid := 1, [1993].log_data[3].valid := 1, [1993].log_data[4].valid := 1, [1993].time.Year := 2022, [1993].time.Month := 4, [1993].time.Day := 30, [1993].time.Hour := 19, [1993].time.Minute := 39, [1993].time.Second := 59, [1993].time.DST_ON := 1, [1994].log_data[0].min := 1.0, [1994].log_data[0].max := 1.0, [1994].log_data[0].total := 300.0, [1994].log_data[0].time := 300.0, [1994].log_data[0].minminute := 40, [1994].log_data[0].maxminute := 40, [1994].log_data[0].valid := 1, [1994].log_data[1].valid := 1, [1994].log_data[2].valid := 1, [1994].log_data[3].valid := 1, [1994].log_data[4].valid := 1, [1994].time.Year := 2022, [1994].time.Month := 4, [1994].time.Day := 30, [1994].time.Hour := 19, [1994].time.Minute := 44, [1994].time.Second := 59, [1994].time.DST_ON := 1, [1995].log_data[0].min := 1.0, [1995].log_data[0].max := 1.0, [1995].log_data[0].total := 300.0, [1995].log_data[0].time := 300.0, [1995].log_data[0].minminute := 45, [1995].log_data[0].maxminute := 45, [1995].log_data[0].valid := 1, [1995].log_data[1].valid := 1, [1995].log_data[2].valid := 1, [1995].log_data[3].valid := 1, [1995].log_data[4].valid := 1, [1995].time.Year := 2022, [1995].time.Month := 4, [1995].time.Day := 30, [1995].time.Hour := 19, [1995].time.Minute := 49, [1995].time.Second := 59, [1995].time.DST_ON := 1, [1996].log_data[0].min := 1.0, [1996].log_data[0].max := 1.0, [1996].log_data[0].total := 300.0,
